C07332=1156.504,165.430,-58.579,-178.413,6.903,148.815
C07333=1156.500,165.680,-58.601,-178.411,6.904,148.815
C07334=1156.495,165.928,-58.623,-178.408,6.906,148.815
C07335=1156.491,166.178,-58.645,-178.405,6.909,148.814
C07336=1156.486,166.426,-58.667,-178.403,6.911,148.814
C07337=1156.481,166.675,-58.690,-178.400,6.913,148.814
C07338=1156.476,166.924,-58.711,-178.397,6.914,148.813
C07339=1156.472,167.173,-58.733,-178.394,6.917,148.813
C07340=1156.467,167.422,-58.755,-178.391,6.919,148.813
C07341=1156.463,167.671,-58.777,-178.389,6.920,148.812
C07342=1156.457,167.920,-58.799,-178.386,6.922,148.812
C07343=1156.453,168.169,-58.821,-178.383,6.925,148.812
C07344=1156.448,168.417,-58.844,-178.380,6.927,148.811
C07345=1156.444,168.667,-58.866,-178.378,6.928,148.811
C07346=1156.438,168.916,-58.888,-178.375,6.930,148.811
C07347=1156.434,169.165,-58.910,-178.372,6.933,148.811
C07348=1156.430,169.414,-58.932,-178.369,6.935,148.810
C07349=1156.425,169.662,-58.955,-178.367,6.937,148.810
C07350=1156.420,169.912,-58.977,-178.364,6.938,148.809
C07351=1156.415,170.161,-58.999,-178.361,6.941,148.809
C07352=1156.411,170.410,-59.021,-178.359,6.943,148.809
C07353=1156.407,170.658,-59.043,-178.356,6.945,148.809
C07354=1156.402,170.908,-59.066,-178.353,6.946,148.808
C07355=1156.397,171.157,-59.088,-178.350,6.949,148.808
C07356=1156.393,171.405,-59.111,-178.347,6.951,148.808
C07357=1156.388,171.655,-59.133,-178.345,6.953,148.807
C07358=1156.383,171.903,-59.155,-178.342,6.955,148.807
C07359=1156.379,172.152,-59.178,-178.339,6.957,148.807
C07360=1156.374,172.402,-59.200,-178.336,6.959,148.806
C07361=1156.369,172.650,-59.222,-178.334,6.961,148.806
C07362=1156.364,172.899,-59.245,-178.331,6.964,148.806
C07363=1156.359,173.148,-59.267,-178.328,6.965,148.805
C07364=1156.355,173.397,-59.290,-178.325,6.967,148.805
C07365=1156.350,173.646,-59.312,-178.322,6.970,148.805
C07366=1156.346,173.895,-59.334,-178.320,6.972,148.805
C07367=1156.341,174.144,-59.357,-178.317,6.973,148.804
C07368=1156.337,174.393,-59.379,-178.315,6.975,148.804
C07369=1156.332,174.642,-59.402,-178.311,6.978,148.803
C07370=1156.327,174.891,-59.425,-178.309,6.980,148.803
C07371=1156.323,175.140,-59.447,-178.306,6.982,148.803
C07372=1156.318,175.389,-59.470,-178.303,6.984,148.803
C07373=1156.314,175.638,-59.492,-178.300,6.986,148.802
C07374=1156.309,175.887,-59.515,-178.298,6.988,148.802
C07375=1156.304,176.135,-59.537,-178.295,6.991,148.802
C07376=1156.299,176.385,-59.560,-178.292,6.992,148.801
C07377=1156.295,176.634,-59.583,-178.290,6.994,148.801
C07378=1156.290,176.882,-59.606,-178.287,6.996,148.801
C07379=1156.285,177.131,-59.628,-178.284,6.999,148.801
C07380=1156.281,177.380,-59.651,-178.281,7.000,148.800
C07381=1156.276,177.630,-59.673,-178.279,7.002,148.800
C07382=1156.271,177.878,-59.696,-178.276,7.005,148.800
C07383=1156.267,178.127,-59.719,-178.273,7.007,148.799
C07384=1156.262,178.376,-59.742,-178.270,7.009,148.799
C07385=1156.258,178.624,-59.764,-178.268,7.012,148.799
C07386=1156.253,178.873,-59.787,-178.265,7.013,148.798
C07387=1156.249,179.123,-59.809,-178.262,7.015,148.798
C07388=1156.244,179.372,-59.833,-178.259,7.018,148.798
C07389=1156.239,179.620,-59.855,-178.257,7.020,148.798
C07390=1156.234,179.869,-59.878,-178.254,7.021,148.797
C07391=1156.230,180.118,-59.901,-178.251,7.024,148.797
C07392=1156.226,180.367,-59.924,-178.249,7.026,148.797
C07393=1156.221,180.616,-59.947,-178.246,7.028,148.796
C07394=1156.216,180.865,-59.969,-178.243,7.030,148.796
C07395=1156.211,181.114,-59.992,-178.240,7.032,148.796
C07396=1156.207,181.363,-60.016,-178.237,7.035,148.796
C07397=1156.203,181.612,-60.038,-178.235,7.037,148.795
C07398=1156.198,181.861,-60.062,-178.232,7.039,148.795
C07399=1156.193,182.110,-60.084,-178.229,7.041,148.795
C07400=1156.189,182.358,-60.107,-178.226,7.043,148.794
C07401=1156.184,182.607,-60.130,-178.224,7.045,148.794
C07402=1156.179,182.856,-60.154,-178.221,7.048,148.794
C07403=1156.175,183.105,-60.176,-178.218,7.050,148.794
C07404=1156.170,183.354,-60.200,-178.215,7.051,148.793
C07405=1156.165,183.624,-60.225,-178.212,7.054,148.793
C07406=1156.161,183.893,-60.249,-178.209,7.057,148.793
C07407=1156.155,184.163,-60.274,-178.207,7.059,148.792
C07408=1156.150,184.433,-60.299,-178.203,7.061,148.792
C07409=1156.145,184.682,-60.323,-178.201,7.063,148.792
C07410=1156.141,184.931,-60.345,-178.198,7.066,148.792
C07411=1156.136,185.179,-60.368,-178.195,7.068,148.791
C07412=1156.131,185.428,-60.392,-178.193,7.069,148.791
C07413=1156.127,185.677,-60.415,-178.190,7.072,148.791
C07414=1156.122,185.926,-60.438,-178.187,7.074,148.790
C07415=1156.118,186.175,-60.461,-178.184,7.077,148.790
C07416=1156.113,186.424,-60.485,-178.182,7.079,148.790
C07417=1156.109,186.673,-60.508,-178.179,7.080,148.790
C07418=1156.104,186.921,-60.532,-178.176,7.083,148.789
C07419=1156.099,187.170,-60.555,-178.173,7.085,148.789
C07420=1156.095,187.419,-60.578,-178.170,7.088,148.789
C07421=1156.090,187.667,-60.601,-178.168,7.089,148.788
C07422=1156.085,187.916,-60.625,-178.165,7.092,148.788
C07423=1156.081,188.165,-60.648,-178.162,7.094,148.788
C07424=1156.076,188.414,-60.671,-178.159,7.096,148.788
C07425=1156.071,188.664,-60.695,-178.157,7.099,148.787
C07426=1156.067,188.913,-60.718,-178.154,7.101,148.787
C07427=1156.062,189.161,-60.742,-178.151,7.102,148.787
C07428=1156.058,189.410,-60.765,-178.148,7.105,148.787
C07429=1156.054,189.659,-60.788,-178.146,7.107,148.786
C07430=1156.049,189.908,-60.811,-178.143,7.110,148.786
C07431=1156.044,190.157,-60.835,-178.140,7.112,148.786
C07432=1156.040,190.405,-60.859,-178.137,7.114,148.785
C07433=1156.035,190.654,-60.882,-178.135,7.116,148.785
C07434=1156.030,190.903,-60.906,-178.132,7.118,148.785
C07435=1156.026,191.152,-60.929,-178.129,7.121,148.785
C07436=1156.021,191.401,-60.953,-178.127,7.123,148.784
C07437=1156.017,191.650,-60.976,-178.123,7.125,148.784
C07438=1156.012,191.899,-61.000,-178.121,7.127,148.784
C07439=1156.008,192.147,-61.024,-178.118,7.129,148.784
C07440=1156.003,192.396,-61.047,-178.115,7.132,148.783
C07441=1155.998,192.645,-61.071,-178.113,7.134,148.783
C07442=1155.994,192.894,-61.095,-178.110,7.136,148.783
C07443=1155.989,193.143,-61.118,-178.107,7.138,148.783
C07444=1155.984,193.392,-61.141,-178.104,7.141,148.782
C07445=1155.980,193.640,-61.165,-178.102,7.143,148.782
C07446=1155.975,193.889,-61.189,-178.099,7.146,148.782
C07447=1155.971,194.138,-61.212,-178.096,7.147,148.782
C07448=1155.966,194.387,-61.236,-178.094,7.150,148.781
C07449=1155.961,194.636,-61.260,-178.091,7.152,148.781
C07450=1155.957,194.884,-61.284,-178.088,7.154,148.781
C07451=1155.952,195.133,-61.307,-178.085,7.157,148.781
C07452=1155.947,195.382,-61.332,-178.082,7.159,148.780
C07453=1155.943,195.632,-61.355,-178.080,7.162,148.780
C07454=1155.939,195.880,-61.380,-178.077,7.163,148.780
C07455=1155.934,196.129,-61.403,-178.074,7.166,148.780
C07456=1155.930,196.377,-61.427,-178.071,7.168,148.779
C07457=1155.925,196.626,-61.450,-178.068,7.171,148.779
C07458=1155.921,196.875,-61.474,-178.066,7.173,148.779
C07459=1155.916,197.124,-61.498,-178.063,7.175,148.779
C07460=1155.911,197.373,-61.522,-178.061,7.177,148.778
C07461=1155.906,197.621,-61.546,-178.058,7.179,148.778
C07462=1155.902,197.871,-61.570,-178.055,7.182,148.778
C07463=1155.898,198.119,-61.594,-178.052,7.184,148.778
C07464=1155.893,198.368,-61.618,-178.049,7.186,148.777
C07465=1155.889,198.617,-61.642,-178.047,7.188,148.777
C07466=1155.884,198.865,-61.666,-178.044,7.191,148.777
C07467=1155.879,199.114,-61.690,-178.041,7.193,148.777
C07468=1155.875,199.363,-61.714,-178.038,7.196,148.776
C07469=1155.871,199.612,-61.738,-178.036,7.198,148.776
C07470=1155.865,199.861,-61.762,-178.033,7.200,148.776
C07471=1155.861,200.110,-61.786,-178.030,7.202,148.776
C07472=1155.856,200.358,-61.810,-178.027,7.205,148.776
C07473=1155.852,200.606,-61.834,-178.025,7.207,148.775
C07474=1155.847,200.857,-61.859,-178.022,7.210,148.775
C07475=1155.843,201.105,-61.883,-178.019,7.211,148.775
C07476=1155.838,201.353,-61.907,-178.016,7.214,148.775
C07477=1155.834,201.602,-61.931,-178.014,7.216,148.774
C07478=1155.829,201.851,-61.955,-178.011,7.219,148.774
C07479=1155.825,202.100,-61.979,-178.008,7.221,148.774
C07480=1155.820,202.349,-62.003,-178.005,7.224,148.774
C07481=1155.815,202.597,-62.028,-178.003,7.226,148.773
C07482=1155.811,202.846,-62.052,-178.000,7.228,148.773
C07483=1155.807,203.095,-62.077,-177.997,7.230,148.773
C07484=1155.802,203.344,-62.101,-177.994,7.233,148.773
C07485=1155.797,203.593,-62.125,-177.992,7.235,148.772
C07486=1155.793,203.841,-62.149,-177.989,7.238,148.772
C07487=1155.788,204.090,-62.174,-177.986,7.240,148.772
C07488=1155.784,204.339,-62.198,-177.983,7.242,148.772
C07489=1155.779,204.588,-62.223,-177.981,7.244,148.772
C07490=1155.774,204.836,-62.247,-177.978,7.247,148.771
C07491=1155.771,205.085,-62.271,-177.975,7.250,148.771
C07492=1155.766,205.334,-62.296,-177.973,7.252,148.771
C07493=1155.761,205.582,-62.320,-177.969,7.254,148.771
C07494=1155.757,205.832,-62.345,-177.967,7.257,148.771
C07495=1155.752,206.080,-62.369,-177.964,7.259,148.770
C07496=1155.747,206.329,-62.394,-177.962,7.261,148.770
C07497=1155.743,206.577,-62.418,-177.958,7.264,148.770
C07498=1155.738,206.827,-62.443,-177.956,7.266,148.770
C07499=1155.734,207.075,-62.467,-177.953,7.269,148.769
C07500=1155.729,207.324,-62.491,-177.951,7.271,148.769
C07501=1155.725,207.573,-62.516,-177.947,7.273,148.769
C07502=1155.720,207.822,-62.541,-177.945,7.275,148.769
C07503=1155.715,208.070,-62.565,-177.942,7.278,148.769
C07504=1155.711,208.319,-62.590,-177.939,7.281,148.768
C07505=1155.706,208.568,-62.614,-177.937,7.283,148.768
C07506=1155.702,208.816,-62.639,-177.934,7.285,148.768
C07507=1155.698,209.065,-62.664,-177.931,7.288,148.768
C07508=1155.693,209.314,-62.688,-177.928,7.290,148.767
C07509=1155.688,209.585,-62.715,-177.925,7.293,148.767
C07510=1155.683,209.855,-62.742,-177.922,7.296,148.767
C07511=1155.678,210.126,-62.769,-177.920,7.298,148.767
C07512=1155.673,210.396,-62.796,-177.917,7.300,148.767
C07513=1155.668,210.645,-62.820,-177.914,7.303,148.767
C07514=1155.664,210.894,-62.845,-177.911,7.305,148.766
C07515=1155.659,211.142,-62.870,-177.908,7.308,148.766
C07516=1155.655,211.391,-62.895,-177.905,7.311,148.766
C07517=1155.651,211.640,-62.919,-177.903,7.313,148.766
C07518=1155.645,211.888,-62.944,-177.900,7.315,148.765
C07519=1155.642,212.137,-62.969,-177.898,7.317,148.765
C07520=1155.637,212.386,-62.994,-177.894,7.320,148.765
C07521=1155.632,212.635,-63.019,-177.891,7.323,148.765
C07522=1155.628,212.883,-63.044,-177.889,7.325,148.765
C07523=1155.624,213.132,-63.069,-177.886,7.328,148.764
C07524=1155.619,213.381,-63.093,-177.884,7.330,148.764
C07525=1155.614,213.630,-63.119,-177.881,7.332,148.764
C07526=1155.610,213.878,-63.143,-177.878,7.334,148.764
C07527=1155.605,214.127,-63.168,-177.876,7.337,148.764
C07528=1155.601,214.376,-63.194,-177.872,7.340,148.763
C07529=1155.596,214.624,-63.218,-177.870,7.342,148.763
C07530=1155.592,214.873,-63.243,-177.867,7.345,148.763
C07531=1155.587,215.122,-63.268,-177.865,7.347,148.763
C07532=1155.583,215.371,-63.294,-177.862,7.350,148.763
C07533=1155.578,215.619,-63.318,-177.859,7.352,148.762
C07534=1155.574,215.868,-63.344,-177.856,7.354,148.762
C07535=1155.569,216.116,-63.368,-177.853,7.357,148.762
C07536=1155.565,216.365,-63.394,-177.850,7.360,148.762
C07537=1155.560,216.614,-63.418,-177.848,7.362,148.762
C07538=1155.556,216.862,-63.444,-177.845,7.365,148.761
C07539=1155.551,217.112,-63.469,-177.843,7.367,148.761
C07540=1155.547,217.360,-63.494,-177.839,7.369,148.761
C07541=1155.542,217.609,-63.520,-177.837,7.372,148.761
C07542=1155.537,217.858,-63.545,-177.834,7.374,148.761
C07543=1155.534,218.106,-63.570,-177.831,7.377,148.761
C07544=1155.529,218.355,-63.595,-177.828,7.380,148.760
C07545=1155.524,218.604,-63.620,-177.826,7.382,148.760
C07546=1155.520,218.852,-63.646,-177.823,7.384,148.760
C07547=1155.515,219.101,-63.671,-177.821,7.387,148.760
C07548=1155.511,219.350,-63.697,-177.818,7.390,148.760
C07549=1155.506,219.598,-63.722,-177.815,7.392,148.759
C07550=1155.501,219.847,-63.747,-177.813,7.394,148.759
C07551=1155.497,220.095,-63.772,-177.809,7.397,148.759
C07552=1155.493,220.344,-63.798,-177.806,7.400,148.759
C07553=1155.489,220.593,-63.823,-177.804,7.402,148.759
C07554=1155.484,220.842,-63.848,-177.801,7.404,148.759
C07555=1155.480,221.090,-63.874,-177.798,7.407,148.758
C07556=1155.475,221.338,-63.899,-177.796,7.409,148.758
C07557=1155.471,221.587,-63.925,-177.793,7.412,148.758
C07558=1155.466,221.837,-63.950,-177.790,7.415,148.758
C07559=1155.461,222.085,-63.975,-177.788,7.417,148.758
C07560=1155.457,222.334,-64.001,-177.785,7.420,148.758
C07561=1155.453,222.582,-64.027,-177.782,7.423,148.757
C07562=1155.448,222.830,-64.052,-177.780,7.425,148.757
C07563=1155.444,223.079,-64.078,-177.776,7.427,148.757
C07564=1155.439,223.329,-64.103,-177.774,7.430,148.757
C07565=1155.434,223.577,-64.128,-177.771,7.432,148.757
C07566=1155.430,223.826,-64.154,-177.768,7.435,148.756
C07567=1155.426,224.074,-64.180,-177.765,7.438,148.756
C07568=1155.421,224.323,-64.205,-177.763,7.440,148.756
C07569=1155.417,224.571,-64.231,-177.760,7.443,148.756
C07570=1155.413,224.820,-64.257,-177.757,7.446,148.756
C07571=1155.407,225.069,-64.283,-177.755,7.448,148.756
C07572=1155.403,225.317,-64.308,-177.752,7.451,148.756
C07573=1155.399,225.566,-64.334,-177.749,7.453,148.755
C07574=1155.394,225.814,-64.360,-177.747,7.455,148.755
C07575=1155.390,226.063,-64.385,-177.744,7.458,148.755
C07576=1155.385,226.312,-64.411,-177.741,7.461,148.755
C07577=1155.381,226.561,-64.437,-177.738,7.464,148.755
C07578=1155.376,226.809,-64.462,-177.736,7.466,148.755
C07579=1155.372,227.058,-64.488,-177.732,7.468,148.754
C07580=1155.367,227.307,-64.514,-177.730,7.471,148.754
C07581=1155.363,227.556,-64.540,-177.727,7.473,148.754
C07582=1155.358,227.804,-64.565,-177.725,7.476,148.754
C07583=1155.354,228.052,-64.592,-177.721,7.479,148.754
C07584=1155.350,228.301,-64.618,-177.719,7.481,148.754
C07585=1155.345,228.550,-64.644,-177.716,7.484,148.754
C07586=1155.340,228.798,-64.669,-177.713,7.487,148.753
C07587=1155.336,229.047,-64.695,-177.710,7.490,148.753
C07588=1155.332,229.295,-64.721,-177.708,7.492,148.753
C07589=1155.328,229.544,-64.747,-177.705,7.495,148.753
C07590=1155.323,229.793,-64.774,-177.702,7.497,148.753
C07591=1155.318,230.041,-64.799,-177.699,7.500,148.753
C07592=1155.314,230.290,-64.825,-177.697,7.502,148.753
C07593=1155.309,230.538,-64.851,-177.694,7.505,148.752
C07594=1155.305,230.787,-64.878,-177.691,7.508,148.752
C07595=1155.301,231.036,-64.903,-177.689,7.510,148.752
C07596=1155.296,231.285,-64.929,-177.686,7.513,148.752
C07597=1155.291,231.532,-64.956,-177.683,7.516,148.752
C07598=1155.287,231.781,-64.982,-177.680,7.518,148.752
C07599=1155.283,232.030,-65.007,-177.678,7.520,148.751
C07600=1155.278,232.278,-65.034,-177.675,7.523,148.751
C07601=1155.274,232.527,-65.060,-177.672,7.526,148.751
C07602=1155.270,232.776,-65.086,-177.669,7.529,148.751
C07603=1155.264,233.024,-65.113,-177.667,7.531,148.751
C07604=1155.260,233.273,-65.138,-177.664,7.534,148.751
C07605=1155.256,233.521,-65.164,-177.661,7.537,148.751
C07606=1155.251,233.770,-65.191,-177.659,7.540,148.751
C07607=1155.247,234.019,-65.217,-177.656,7.542,148.750
C07608=1155.242,234.267,-65.244,-177.653,7.545,148.750
C07609=1155.238,234.516,-65.270,-177.650,7.547,148.750
C07610=1155.234,234.764,-65.296,-177.648,7.550,148.750
C07611=1155.229,235.013,-65.323,-177.645,7.552,148.750
C07612=1155.225,235.262,-65.349,-177.642,7.555,148.750
C07613=1155.220,235.534,-65.378,-177.639,7.558,148.750
C07614=1155.215,235.805,-65.406,-177.637,7.561,148.749
C07615=1155.210,236.077,-65.435,-177.633,7.564,148.749
C07616=1155.206,236.349,-65.464,-177.630,7.567,148.749
C07617=1155.201,236.597,-65.491,-177.628,7.569,148.749
C07618=1155.197,236.846,-65.517,-177.625,7.572,148.749
C07619=1155.192,237.094,-65.544,-177.622,7.575,148.749
C07620=1155.188,237.343,-65.569,-177.619,7.578,148.749
C07621=1155.183,237.592,-65.596,-177.616,7.581,148.749
C07622=1155.179,237.840,-65.623,-177.614,7.583,148.748
C07623=1155.174,238.089,-65.649,-177.611,7.586,148.748
C07624=1155.170,238.337,-65.676,-177.608,7.589,148.748
C07625=1155.166,238.586,-65.703,-177.605,7.591,148.748
C07626=1155.161,238.835,-65.729,-177.603,7.594,148.748
C07627=1155.157,239.083,-65.756,-177.600,7.596,148.748
C07628=1155.152,239.331,-65.783,-177.597,7.599,148.748
C07629=1155.148,239.580,-65.808,-177.595,7.602,148.748
C07630=1155.143,239.829,-65.835,-177.591,7.605,148.747
C07631=1155.139,240.077,-65.862,-177.589,7.607,148.747
C07632=1155.135,240.325,-65.889,-177.586,7.610,148.747
C07633=1155.130,240.574,-65.916,-177.584,7.613,148.747
C07634=1155.126,240.823,-65.942,-177.581,7.616,148.747
C07635=1155.121,241.071,-65.969,-177.578,7.619,148.747
C07636=1155.117,241.320,-65.996,-177.575,7.621,148.747
C07637=1155.113,241.568,-66.022,-177.573,7.624,148.747
C07638=1155.108,241.816,-66.049,-177.570,7.626,148.746
C07639=1155.103,242.065,-66.076,-177.567,7.629,148.746
C07640=1155.099,242.314,-66.102,-177.564,7.632,148.746
C07641=1155.094,242.562,-66.129,-177.562,7.635,148.746
C07642=1155.090,242.811,-66.156,-177.559,7.637,148.746
C07643=1155.086,243.059,-66.183,-177.556,7.640,148.746
C07644=1155.081,243.307,-66.210,-177.553,7.643,148.746
C07645=1155.077,243.556,-66.237,-177.551,7.646,148.746
C07646=1155.073,243.804,-66.263,-177.548,7.649,148.746
C07647=1155.069,244.053,-66.291,-177.546,7.651,148.746
C07648=1155.064,244.302,-66.318,-177.543,7.654,148.745
C07649=1155.059,244.550,-66.345,-177.540,7.657,148.745
C07650=1155.055,244.798,-66.371,-177.537,7.660,148.745
C07651=1155.051,245.047,-66.399,-177.534,7.663,148.745
C07652=1155.046,245.295,-66.426,-177.531,7.665,148.745
C07653=1155.041,245.544,-66.453,-177.529,7.667,148.745
C07654=1155.037,245.792,-66.479,-177.526,7.670,148.745
C07655=1155.033,246.041,-66.507,-177.523,7.673,148.745
C07656=1155.029,246.290,-66.534,-177.521,7.676,148.745
C07657=1155.024,246.538,-66.561,-177.518,7.679,148.745
C07658=1155.019,246.787,-66.588,-177.515,7.682,148.744
C07659=1155.015,247.035,-66.615,-177.512,7.685,148.744
C07660=1155.011,247.283,-66.641,-177.510,7.687,148.744
C07661=1155.007,247.532,-66.669,-177.507,7.690,148.744
C07662=1155.002,247.781,-66.696,-177.504,7.693,148.744
C07663=1154.998,248.029,-66.724,-177.501,7.696,148.744
C07664=1154.993,248.277,-66.751,-177.499,7.699,148.744
C07665=1154.989,248.526,-66.778,-177.496,7.702,148.744
C07666=1154.984,248.774,-66.805,-177.494,7.704,148.744
C07667=1154.980,249.023,-66.833,-177.491,7.707,148.744
C07668=1154.975,249.272,-66.860,-177.488,7.709,148.744
C07669=1154.972,249.520,-66.886,-177.485,7.712,148.743
C07670=1154.967,249.768,-66.913,-177.483,7.715,148.743
C07671=1154.963,250.017,-66.942,-177.480,7.718,148.743
C07672=1154.958,250.265,-66.969,-177.477,7.721,148.743
C07673=1154.954,250.514,-66.996,-177.474,7.724,148.743
C07674=1154.949,250.762,-67.023,-177.472,7.726,148.743
C07675=1154.945,251.011,-67.051,-177.469,7.729,148.743
C07676=1154.941,251.259,-67.078,-177.466,7.732,148.743
C07677=1154.936,251.507,-67.106,-177.464,7.735,148.743
C07678=1154.932,251.756,-67.133,-177.460,7.738,148.743
C07679=1154.928,252.005,-67.160,-177.458,7.741,148.743
C07680=1154.923,252.253,-67.188,-177.455,7.744,148.742
C07681=1154.919,252.501,-67.215,-177.452,7.747,148.742
C07682=1154.914,252.749,-67.243,-177.450,7.749,148.742
C07683=1154.910,252.998,-67.270,-177.447,7.752,148.742
C07684=1154.906,253.247,-67.297,-177.444,7.755,148.742
C07685=1154.901,253.495,-67.325,-177.442,7.757,148.742
C07686=1154.897,253.744,-67.353,-177.439,7.760,148.742
C07687=1154.893,253.992,-67.380,-177.436,7.763,148.742
C07688=1154.887,254.241,-67.408,-177.433,7.766,148.742
C07689=1154.884,254.489,-67.436,-177.431,7.769,148.742
C07690=1154.879,254.738,-67.463,-177.428,7.772,148.742
C07691=1154.875,254.986,-67.491,-177.426,7.774,148.742
C07692=1154.871,255.234,-67.519,-177.423,7.777,148.742
C07693=1154.866,255.483,-67.546,-177.420,7.780,148.742
C07694=1154.862,255.731,-67.574,-177.417,7.783,148.741
C07695=1154.858,255.980,-67.601,-177.414,7.786,148.741
C07696=1154.853,256.228,-67.630,-177.412,7.789,148.741
C07697=1154.848,256.476,-67.657,-177.409,7.792,148.741
C07698=1154.844,256.725,-67.685,-177.406,7.795,148.741
C07699=1154.840,256.973,-67.713,-177.403,7.798,148.741
C07700=1154.836,257.222,-67.740,-177.401,7.801,148.741
C07701=1154.832,257.470,-67.768,-177.398,7.804,148.741
C07702=1154.827,257.718,-67.796,-177.396,7.806,148.741
C07703=1154.822,257.967,-67.824,-177.393,7.809,148.741
C07704=1154.818,258.215,-67.852,-177.390,7.812,148.741
C07705=1154.814,258.464,-67.880,-177.387,7.815,148.741
C07706=1154.809,258.712,-67.908,-177.385,7.818,148.741
C07707=1154.805,258.960,-67.935,-177.382,7.821,148.741
C07708=1154.801,259.209,-67.963,-177.379,7.823,148.741
C07709=1154.797,259.457,-67.991,-177.377,7.827,148.741
C07710=1154.792,259.706,-68.020,-177.374,7.830,148.741
C07711=1154.788,259.954,-68.048,-177.371,7.833,148.741
C07712=1154.784,260.203,-68.075,-177.368,7.836,148.741
C07713=1154.779,260.451,-68.103,-177.366,7.839,148.740
C07714=1154.774,260.699,-68.131,-177.363,7.841,148.740
C07715=1154.770,260.947,-68.159,-177.360,7.844,148.740
C07716=1154.766,261.195,-68.187,-177.358,7.847,148.740
C07717=1154.761,261.469,-68.218,-177.355,7.850,148.740
C07718=1154.756,261.742,-68.249,-177.352,7.853,148.740
C07719=1154.751,262.016,-68.280,-177.349,7.856,148.740
C07720=1154.747,262.289,-68.310,-177.346,7.860,148.740
C07721=1154.742,262.538,-68.339,-177.343,7.863,148.740
C07722=1154.738,262.786,-68.367,-177.340,7.866,148.740
C07723=1154.733,263.035,-68.396,-177.337,7.869,148.740
C07724=1154.729,263.283,-68.423,-177.335,7.872,148.740
C07725=1154.725,263.531,-68.452,-177.332,7.875,148.740
C07726=1154.720,263.779,-68.480,-177.329,7.878,148.740
C07727=1154.716,264.028,-68.508,-177.327,7.880,148.740
C07728=1154.712,264.277,-68.537,-177.324,7.883,148.740
C07729=1154.708,264.525,-68.565,-177.322,7.886,148.740
C07730=1154.703,264.774,-68.593,-177.319,7.889,148.740
C07731=1154.699,265.021,-68.622,-177.316,7.892,148.740
C07732=1154.695,265.270,-68.651,-177.313,7.895,148.740
C07733=1154.690,265.518,-68.678,-177.311,7.898,148.740
C07734=1154.686,265.766,-68.707,-177.308,7.901,148.739
C07735=1154.681,266.014,-68.735,-177.305,7.904,148.739
C07736=1154.677,266.263,-68.764,-177.302,7.907,148.739
C07737=1154.673,266.512,-68.792,-177.300,7.910,148.740
C07738=1154.668,266.760,-68.820,-177.297,7.913,148.739
C07739=1154.665,267.008,-68.849,-177.294,7.916,148.739
C07740=1154.660,267.256,-68.877,-177.292,7.919,148.739
C07741=1154.656,267.505,-68.905,-177.289,7.922,148.739
C07742=1154.651,267.753,-68.934,-177.286,7.925,148.739
C07743=1154.647,268.001,-68.963,-177.283,7.927,148.739
C07744=1154.643,268.250,-68.991,-177.281,7.930,148.739
C07745=1154.638,268.498,-69.020,-177.278,7.934,148.739
C07746=1154.634,268.746,-69.048,-177.276,7.937,148.739
C07747=1154.630,268.995,-69.077,-177.273,7.940,148.739
C07748=1154.625,269.243,-69.105,-177.270,7.943,148.739
C07749=1154.621,269.492,-69.134,-177.267,7.945,148.739
C07750=1154.617,269.740,-69.163,-177.264,7.948,148.739
C07751=1154.612,269.988,-69.191,-177.262,7.952,148.739
C07752=1154.608,270.237,-69.220,-177.259,7.955,148.739
C07753=1154.604,270.485,-69.249,-177.257,7.958,148.739
C07754=1154.599,270.733,-69.277,-177.254,7.961,148.739
C07755=1154.595,270.981,-69.307,-177.251,7.963,148.739
C07756=1154.591,271.230,-69.335,-177.248,7.966,148.739
C07757=1154.586,271.478,-69.363,-177.246,7.970,148.739
C07758=1154.582,271.726,-69.392,-177.243,7.973,148.739
C07759=1154.578,271.975,-69.421,-177.240,7.976,148.739
C07760=1154.574,272.222,-69.450,-177.238,7.979,148.739
C07761=1154.569,272.471,-69.478,-177.235,7.981,148.739
C07762=1154.565,272.719,-69.508,-177.233,7.985,148.739
C07763=1154.560,272.968,-69.537,-177.230,7.988,148.739
C07764=1154.556,273.215,-69.565,-177.227,7.991,148.739
C07765=1154.552,273.464,-69.594,-177.224,7.994,148.739
C07766=1154.548,273.713,-69.623,-177.221,7.997,148.739
C07767=1154.543,273.961,-69.652,-177.219,8.000,148.739
C07768=1154.539,274.209,-69.681,-177.216,8.003,148.739
C07769=1154.535,274.457,-69.710,-177.214,8.006,148.739
C07770=1154.531,274.706,-69.739,-177.211,8.009,148.739
C07771=1154.526,274.954,-69.768,-177.208,8.012,148.739
C07772=1154.521,275.202,-69.797,-177.206,8.015,148.739
C07773=1154.518,275.450,-69.825,-177.203,8.018,148.739
C07774=1154.514,275.699,-69.855,-177.200,8.021,148.739
C07775=1154.509,275.947,-69.884,-177.197,8.024,148.739
C07776=1154.504,276.195,-69.913,-177.195,8.027,148.739
C07777=1154.500,276.443,-69.942,-177.192,8.030,148.739
C07778=1154.496,276.692,-69.972,-177.190,8.033,148.739
C07779=1154.492,276.940,-70.000,-177.187,8.036,148.739
C07780=1154.488,277.188,-70.029,-177.185,8.039,148.739
C07781=1154.483,277.436,-70.058,-177.182,8.042,148.739
C07782=1154.479,277.684,-70.088,-177.179,8.045,148.739
C07783=1154.475,277.933,-70.116,-177.176,8.048,148.739
C07784=1154.470,278.181,-70.146,-177.174,8.051,148.739
C07785=1154.466,278.430,-70.175,-177.171,8.055,148.739
C07786=1154.462,278.678,-70.205,-177.168,8.058,148.739
C07787=1154.458,278.926,-70.234,-177.165,8.061,148.739
C07788=1154.453,279.174,-70.263,-177.163,8.064,148.739
C07789=1154.449,279.423,-70.292,-177.160,8.067,148.739
C07790=1154.444,279.671,-70.322,-177.157,8.070,148.739
C07791=1154.440,279.919,-70.351,-177.154,8.073,148.739
C07792=1154.436,280.167,-70.380,-177.152,8.076,148.739
C07793=1154.432,280.416,-70.410,-177.149,8.079,148.739
C07794=1154.428,280.664,-70.439,-177.147,8.082,148.739
C07795=1154.424,280.912,-70.469,-177.144,8.085,148.739
C07796=1154.419,281.160,-70.498,-177.142,8.088,148.739
C07797=1154.415,281.408,-70.527,-177.139,8.091,148.739
C07798=1154.410,281.656,-70.557,-177.136,8.095,148.739
C07799=1154.406,281.905,-70.586,-177.134,8.098,148.739
C07800=1154.402,282.153,-70.616,-177.131,8.101,148.739
C07801=1154.398,282.401,-70.645,-177.128,8.103,148.739
C07802=1154.394,282.649,-70.675,-177.126,8.107,148.739
C07803=1154.390,282.898,-70.704,-177.122,8.111,148.739
C07804=1154.385,283.146,-70.734,-177.120,8.113,148.739
C07805=1154.380,283.395,-70.764,-177.117,8.117,148.739
C07806=1154.376,283.643,-70.793,-177.115,8.120,148.739
C07807=1154.372,283.891,-70.823,-177.112,8.123,148.739
C07808=1154.368,284.139,-70.852,-177.110,8.126,148.739
C07809=1154.364,284.387,-70.882,-177.107,8.129,148.739
C07810=1154.360,284.635,-70.912,-177.104,8.132,148.739
C07811=1154.356,284.884,-70.941,-177.102,8.135,148.740
C07812=1154.350,285.131,-70.971,-177.099,8.138,148.740
C07813=1154.346,285.380,-71.000,-177.096,8.141,148.739
C07814=1154.342,285.628,-71.030,-177.094,8.144,148.740
C07815=1154.338,285.876,-71.060,-177.091,8.148,148.740
C07816=1154.334,286.124,-71.089,-177.088,8.151,148.740
C07817=1154.329,286.372,-71.119,-177.085,8.154,148.740
C07818=1154.325,286.621,-71.149,-177.083,8.157,148.740
C07819=1154.321,286.869,-71.179,-177.080,8.160,148.740
C07820=1154.317,287.117,-71.209,-177.078,8.163,148.740
C07821=1154.312,287.392,-71.242,-177.074,8.167,148.740
C07822=1154.308,287.667,-71.275,-177.072,8.170,148.740
C07823=1154.303,287.942,-71.308,-177.069,8.174,148.740
C07824=1154.297,288.218,-71.341,-177.066,8.177,148.740
C07825=1154.293,288.466,-71.371,-177.064,8.180,148.740
C07826=1154.289,288.714,-71.401,-177.061,8.183,148.740
C07827=1154.285,288.962,-71.430,-177.058,8.186,148.740
C07828=1154.281,289.211,-71.461,-177.055,8.190,148.740
C07829=1154.277,289.459,-71.491,-177.052,8.193,148.740
C07830=1154.273,289.707,-71.521,-177.050,8.197,148.740
C07831=1154.268,289.955,-71.551,-177.047,8.200,148.740
C07832=1154.264,290.203,-71.581,-177.044,8.203,148.740
C07833=1154.260,290.451,-71.611,-177.042,8.206,148.741
C07834=1154.255,290.700,-71.641,-177.039,8.209,148.740
C07835=1154.251,290.947,-71.671,-177.037,8.212,148.741
C07836=1154.247,291.195,-71.702,-177.034,8.215,148.741
C07837=1154.242,291.444,-71.731,-177.031,8.219,148.741
C07838=1154.239,291.692,-71.762,-177.029,8.222,148.741
C07839=1154.234,291.941,-71.792,-177.026,8.225,148.741
C07840=1154.230,292.188,-71.822,-177.024,8.228,148.741
C07841=1154.225,292.437,-71.852,-177.021,8.231,148.741
C07842=1154.221,292.684,-71.882,-177.019,8.235,148.741
C07843=1154.218,292.932,-71.912,-177.016,8.237,148.741
C07844=1154.213,293.181,-71.943,-177.013,8.241,148.741
C07845=1154.209,293.429,-71.973,-177.010,8.245,148.741
C07846=1154.205,293.678,-72.003,-177.008,8.248,148.741
C07847=1154.201,293.925,-72.033,-177.005,8.251,148.741
C07848=1154.196,294.173,-72.064,-177.002,8.254,148.741
C07849=1154.192,294.421,-72.094,-177.000,8.257,148.741
C07850=1154.188,294.670,-72.124,-176.997,8.260,148.741
C07851=1154.184,294.918,-72.155,-176.995,8.263,148.742
C07852=1154.179,295.166,-72.185,-176.992,8.267,148.742
C07853=1154.175,295.414,-72.215,-176.989,8.270,148.742
C07854=1154.171,295.662,-72.246,-176.986,8.273,148.742
C07855=1154.167,295.910,-72.276,-176.984,8.276,148.742
C07856=1154.163,296.158,-72.307,-176.981,8.279,148.742
C07857=1154.158,296.406,-72.338,-176.979,8.283,148.742
C07858=1154.154,296.654,-72.367,-176.976,8.286,148.742
C07859=1154.150,296.903,-72.398,-176.973,8.290,148.742
C07860=1154.146,297.151,-72.428,-176.971,8.293,148.742
C07861=1154.141,297.399,-72.459,-176.968,8.296,148.742
C07862=1154.137,297.647,-72.490,-176.966,8.299,148.742
C07863=1154.133,297.895,-72.520,-176.963,8.302,148.743
C07864=1154.129,298.143,-72.551,-176.960,8.305,148.743
C07865=1154.125,298.391,-72.581,-176.958,8.309,148.743
C07866=1154.120,298.639,-72.611,-176.955,8.312,148.743
C07867=1154.116,298.888,-72.643,-176.953,8.315,148.743
C07868=1154.112,299.136,-72.673,-176.950,8.318,148.743
C07869=1154.108,299.383,-72.703,-176.947,8.322,148.743
C07870=1154.104,299.632,-72.735,-176.945,8.325,148.743
C07871=1154.100,299.880,-72.765,-176.942,8.329,148.743
C07872=1154.095,300.128,-72.796,-176.939,8.332,148.743
C07873=1154.090,300.376,-72.826,-176.937,8.335,148.743
C07874=1154.086,300.624,-72.857,-176.934,8.338,148.744
C07875=1154.083,300.872,-72.888,-176.932,8.341,148.744
C07876=1154.078,301.119,-72.919,-176.929,8.344,148.744
C07877=1154.074,301.368,-72.950,-176.926,8.348,148.744
C07878=1154.070,301.616,-72.981,-176.924,8.352,148.744
C07879=1154.066,301.864,-73.011,-176.921,8.354,148.744
C07880=1154.062,302.112,-73.042,-176.919,8.358,148.744
C07881=1154.057,302.360,-73.073,-176.916,8.361,148.744
C07882=1154.053,302.609,-73.104,-176.913,8.365,148.744
C07883=1154.048,302.857,-73.135,-176.911,8.368,148.744
C07884=1154.045,303.104,-73.166,-176.908,8.371,148.744
C07885=1154.041,303.353,-73.197,-176.906,8.374,148.745
C07886=1154.036,303.600,-73.228,-176.903,8.378,148.745
C07887=1154.032,303.848,-73.258,-176.900,8.381,148.745
C07888=1154.028,304.097,-73.290,-176.898,8.385,148.745
C07889=1154.023,304.344,-73.321,-176.895,8.388,148.745
C07890=1154.019,304.593,-73.352,-176.892,8.391,148.745
C07891=1154.015,304.841,-73.382,-176.890,8.394,148.745
C07892=1154.011,305.089,-73.413,-176.887,8.398,148.745
C07893=1154.007,305.337,-73.445,-176.885,8.401,148.745
C07894=1154.003,305.585,-73.476,-176.882,8.404,148.745
C07895=1153.999,305.833,-73.507,-176.879,8.407,148.746
C07896=1153.994,306.081,-73.538,-176.877,8.411,148.746
C07897=1153.990,306.329,-73.569,-176.874,8.414,148.746
C07898=1153.986,306.577,-73.601,-176.871,8.418,148.746
C07899=1153.981,306.825,-73.632,-176.869,8.421,148.746
C07900=1153.977,307.073,-73.663,-176.866,8.424,148.746
C07901=1153.973,307.321,-73.694,-176.864,8.427,148.746
C07902=1153.969,307.569,-73.725,-176.861,8.431,148.746
C07903=1153.965,307.817,-73.757,-176.858,8.434,148.747
C07904=1153.961,308.065,-73.788,-176.856,8.438,148.747
C07905=1153.956,308.313,-73.820,-176.853,8.441,148.747
C07906=1153.952,308.561,-73.851,-176.851,8.444,148.747
C07907=1153.948,308.809,-73.882,-176.848,8.448,148.747
C07908=1153.944,309.057,-73.913,-176.845,8.451,148.747
C07909=1153.940,309.305,-73.945,-176.843,8.454,148.747
C07910=1153.936,309.553,-73.976,-176.841,8.457,148.747
C07911=1153.931,309.801,-74.007,-176.837,8.461,148.747
C07912=1153.927,310.049,-74.039,-176.835,8.464,148.748
C07913=1153.923,310.297,-74.070,-176.833,8.468,148.748
C07914=1153.919,310.545,-74.101,-176.830,8.471,148.748
C07915=1153.915,310.793,-74.133,-176.827,8.475,148.748
C07916=1153.911,311.041,-74.164,-176.825,8.478,148.748
C07917=1153.906,311.289,-74.195,-176.822,8.481,148.748
C07918=1153.903,311.537,-74.227,-176.820,8.484,148.748
C07919=1153.898,311.784,-74.259,-176.817,8.488,148.749
C07920=1153.894,312.033,-74.290,-176.814,8.491,148.749
C07921=1153.890,312.281,-74.322,-176.812,8.495,148.749
C07922=1153.886,312.528,-74.354,-176.809,8.498,148.749
C07923=1153.882,312.777,-74.385,-176.807,8.502,148.749
C07924=1153.877,313.024,-74.416,-176.804,8.505,148.749
C07925=1153.873,313.302,-74.452,-176.801,8.509,148.749
C07926=1153.869,313.579,-74.487,-176.799,8.512,148.750
C07927=1153.863,313.857,-74.523,-176.795,8.516,148.750
C07928=1153.858,314.135,-74.558,-176.792,8.520,148.750
C07929=1153.855,314.383,-74.590,-176.790,8.523,148.750
C07930=1153.850,314.630,-74.621,-176.788,8.527,148.750
C07931=1153.847,314.878,-74.653,-176.784,8.531,148.750
C07932=1153.842,315.126,-74.686,-176.782,8.534,148.750
C07933=1153.838,315.374,-74.717,-176.780,8.537,148.751
C07934=1153.834,315.622,-74.749,-176.777,8.540,148.751
C07935=1153.830,315.870,-74.780,-176.774,8.544,148.751
C07936=1153.825,316.118,-74.812,-176.772,8.547,148.751
C07937=1153.821,316.366,-74.844,-176.769,8.551,148.751
C07938=1153.817,316.613,-74.876,-176.767,8.554,148.751
C07939=1153.813,316.862,-74.907,-176.764,8.558,148.751
C07940=1153.809,317.110,-74.940,-176.762,8.561,148.752
C07941=1153.805,317.358,-74.972,-176.759,8.564,148.752
C07942=1153.801,317.605,-75.003,-176.756,8.568,148.752
C07943=1153.797,317.854,-75.036,-176.754,8.571,148.752
C07944=1153.793,318.102,-75.068,-176.751,8.575,148.752
C07945=1153.789,318.349,-75.099,-176.749,8.578,148.752
C07946=1153.784,318.597,-75.131,-176.746,8.582,148.753
C07947=1153.780,318.845,-75.163,-176.744,8.585,148.753
C07948=1153.776,319.093,-75.195,-176.741,8.588,148.753
C07949=1153.772,319.340,-75.228,-176.738,8.592,148.753
C07950=1153.768,319.588,-75.260,-176.736,8.596,148.753
C07951=1153.764,319.837,-75.292,-176.733,8.599,148.753
C07952=1153.759,320.084,-75.324,-176.731,8.602,148.754
C07953=1153.756,320.332,-75.356,-176.728,8.606,148.754
C07954=1153.751,320.581,-75.388,-176.725,8.609,148.754
C07955=1153.748,320.828,-75.421,-176.723,8.612,148.754
C07956=1153.743,321.076,-75.453,-176.720,8.617,148.754
C07957=1153.739,321.324,-75.484,-176.718,8.620,148.754
C07958=1153.735,321.572,-75.517,-176.716,8.623,148.755
C07959=1153.731,321.820,-75.549,-176.712,8.627,148.755
C07960=1153.727,322.068,-75.582,-176.710,8.630,148.755
C07961=1153.723,322.315,-75.613,-176.708,8.633,148.755
C07962=1153.718,322.563,-75.646,-176.705,8.637,148.755
C07963=1153.715,322.811,-75.678,-176.702,8.641,148.755
C07964=1153.710,323.059,-75.711,-176.700,8.644,148.756
C07965=1153.707,323.307,-75.743,-176.698,8.647,148.756
C07966=1153.702,323.556,-75.775,-176.694,8.651,148.756
C07967=1153.698,323.802,-75.807,-176.692,8.654,148.756
C07968=1153.694,324.051,-75.840,-176.690,8.658,148.756
C07969=1153.690,324.298,-75.872,-176.687,8.662,148.757
C07970=1153.686,324.546,-75.905,-176.685,8.665,148.757
C07971=1153.682,324.795,-75.937,-176.682,8.668,148.757
C07972=1153.678,325.042,-75.970,-176.679,8.672,148.757
C07973=1153.673,325.290,-76.002,-176.677,8.676,148.757
C07974=1153.670,325.537,-76.034,-176.674,8.679,148.757
C07975=1153.665,325.786,-76.067,-176.671,8.683,148.758
C07976=1153.662,326.033,-76.099,-176.669,8.686,148.758
C07977=1153.657,326.281,-76.132,-176.667,8.689,148.758
C07978=1153.653,326.529,-76.165,-176.664,8.693,148.758
C07979=1153.649,326.777,-76.197,-176.662,8.697,148.758
C07980=1153.645,327.025,-76.230,-176.659,8.700,148.759
C07981=1153.640,327.273,-76.262,-176.656,8.704,148.759
C07982=1153.637,327.520,-76.295,-176.654,8.707,148.759
C07983=1153.632,327.768,-76.327,-176.652,8.711,148.759
C07984=1153.628,328.016,-76.360,-176.649,8.715,148.759
C07985=1153.625,328.263,-76.393,-176.647,8.718,148.760
C07986=1153.620,328.512,-76.425,-176.644,8.721,148.760
C07987=1153.616,328.760,-76.458,-176.641,8.725,148.760
C07988=1153.612,329.007,-76.492,-176.639,8.728,148.760
C07989=1153.608,329.255,-76.523,-176.636,8.732,148.760
C07990=1153.604,329.503,-76.557,-176.633,8.736,148.760
C07991=1153.600,329.751,-76.590,-176.631,8.739,148.761
C07992=1153.596,329.999,-76.622,-176.628,8.743,148.761
C07993=1153.592,330.247,-76.655,-176.626,8.746,148.761
C07994=1153.588,330.494,-76.688,-176.624,8.750,148.761
C07995=1153.584,330.742,-76.721,-176.621,8.754,148.762
C07996=1153.580,330.990,-76.753,-176.618,8.757,148.762
C07997=1153.575,331.238,-76.787,-176.616,8.760,148.762
C07998=1153.572,331.486,-76.819,-176.613,8.764,148.762
C07999=1153.568,331.733,-76.852,-176.611,8.768,148.762
C08000=1153.563,331.982,-76.885,-176.608,8.772,148.763
C08001=1153.559,332.229,-76.918,-176.606,8.775,148.763
C08002=1153.555,332.477,-76.951,-176.603,8.778,148.763
C08003=1153.551,332.725,-76.984,-176.600,8.782,148.763
C08004=1153.547,332.973,-77.017,-176.598,8.786,148.763
C08005=1153.543,333.220,-77.051,-176.596,8.789,148.764
C08006=1153.539,333.468,-77.083,-176.593,8.793,148.764
C08007=1153.535,333.715,-77.116,-176.591,8.796,148.764
C08008=1153.531,333.963,-77.149,-176.588,8.800,148.764
C08009=1153.527,334.211,-77.183,-176.585,8.804,148.765
C08010=1153.523,334.459,-77.216,-176.583,8.807,148.765
C08011=1153.518,334.707,-77.248,-176.580,8.811,148.765
C08012=1153.514,334.955,-77.281,-176.578,8.814,148.765
C08013=1153.510,335.202,-77.314,-176.575,8.818,148.765
C08014=1153.506,335.449,-77.348,-176.573,8.822,148.766
C08015=1153.502,335.697,-77.381,-176.570,8.825,148.766
C08016=1153.498,335.945,-77.415,-176.567,8.829,148.766
C08017=1153.494,336.193,-77.448,-176.565,8.832,148.766
C08018=1153.490,336.440,-77.481,-176.563,8.836,148.767
C08019=1153.486,336.689,-77.514,-176.560,8.840,148.767
C08020=1153.482,336.937,-77.548,-176.558,8.843,148.767
C08021=1153.478,337.184,-77.581,-176.555,8.847,148.767
C08022=1153.474,337.432,-77.614,-176.552,8.850,148.767
C08023=1153.470,337.680,-77.647,-176.549,8.854,148.768
C08024=1153.466,337.927,-77.681,-176.548,8.858,148.768
C08025=1153.462,338.175,-77.714,-176.545,8.861,148.768
C08026=1153.458,338.422,-77.747,-176.542,8.865,148.769
C08027=1153.454,338.671,-77.781,-176.540,8.869,148.769
C08028=1153.450,338.918,-77.814,-176.537,8.873,148.769
C08029=1153.445,339.198,-77.852,-176.534,8.877,148.769
C08030=1153.441,339.479,-77.890,-176.531,8.881,148.769
C08031=1153.436,339.758,-77.927,-176.528,8.885,148.770
C08032=1153.431,340.039,-77.966,-176.525,8.889,148.770
C08033=1153.427,340.287,-77.999,-176.523,8.892,148.770
C08034=1153.423,340.534,-78.033,-176.521,8.897,148.771
C08035=1153.419,340.781,-78.066,-176.518,8.900,148.771
C08036=1153.415,341.029,-78.099,-176.516,8.903,148.771
C08037=1153.411,341.276,-78.133,-176.513,8.908,148.771
C08038=1153.407,341.525,-78.167,-176.511,8.911,148.771
C08039=1153.403,341.772,-78.201,-176.508,8.915,148.772
C08040=1153.399,342.020,-78.234,-176.506,8.918,148.772
C08041=1153.395,342.268,-78.267,-176.503,8.922,148.772
C08042=1153.391,342.516,-78.302,-176.500,8.926,148.772
C08043=1153.387,342.763,-78.335,-176.499,8.929,148.773
C08044=1153.383,343.011,-78.369,-176.496,8.933,148.773
C08045=1153.379,343.258,-78.403,-176.493,8.937,148.773
C08046=1153.374,343.506,-78.437,-176.490,8.941,148.774
C08047=1153.371,343.754,-78.471,-176.488,8.944,148.774
C08048=1153.367,344.001,-78.504,-176.485,8.948,148.774
C08049=1153.363,344.249,-78.538,-176.483,8.952,148.774
C08050=1153.358,344.496,-78.572,-176.480,8.956,148.775
C08051=1153.354,344.745,-78.606,-176.478,8.959,148.775
C08052=1153.351,344.992,-78.639,-176.475,8.963,148.775
C08053=1153.346,345.240,-78.673,-176.473,8.966,148.775
C08054=1153.343,345.488,-78.707,-176.470,8.970,148.776
C08055=1153.339,345.735,-78.741,-176.468,8.974,148.776
C08056=1153.334,345.983,-78.775,-176.466,8.977,148.776
C08057=1153.330,346.230,-78.809,-176.463,8.981,148.776
C08058=1153.327,346.478,-78.843,-176.461,8.985,148.777
C08059=1153.322,346.726,-78.877,-176.458,8.989,148.777
C08060=1153.318,346.973,-78.911,-176.456,8.992,148.777
C08061=1153.314,347.221,-78.946,-176.453,8.996,148.778
C08062=1153.310,347.469,-78.979,-176.451,9.000,148.778
C08063=1153.306,347.716,-79.013,-176.448,9.004,148.778
C08064=1153.302,347.964,-79.047,-176.445,9.007,148.778
C08065=1153.298,348.211,-79.081,-176.443,9.011,148.779
C08066=1153.293,348.459,-79.115,-176.441,9.015,148.779
C08067=1153.290,348.707,-79.149,-176.438,9.019,148.779
C08068=1153.286,348.954,-79.184,-176.435,9.022,148.779
C08069=1153.282,349.202,-79.218,-176.433,9.027,148.780
C08070=1153.278,349.450,-79.252,-176.431,9.030,148.780
C08071=1153.274,349.697,-79.286,-176.428,9.034,148.780
C08072=1153.270,349.946,-79.320,-176.425,9.037,148.780
C08073=1153.266,350.193,-79.354,-176.422,9.041,148.781
C08074=1153.262,350.441,-79.389,-176.421,9.045,148.781
C08075=1153.258,350.688,-79.423,-176.418,9.049,148.781
C08076=1153.254,350.935,-79.457,-176.415,9.052,148.782
C08077=1153.250,351.183,-79.492,-176.413,9.057,148.782
C08078=1153.246,351.430,-79.526,-176.411,9.060,148.782
C08079=1153.242,351.678,-79.560,-176.408,9.064,148.783
C08080=1153.238,351.926,-79.595,-176.405,9.067,148.783
C08081=1153.235,352.174,-79.629,-176.403,9.072,148.783
C08082=1153.230,352.421,-79.664,-176.401,9.075,148.783
C08083=1153.226,352.668,-79.698,-176.398,9.079,148.784
C08084=1153.222,352.916,-79.732,-176.395,9.082,148.784
C08085=1153.218,353.164,-79.767,-176.393,9.087,148.784
C08086=1153.215,353.411,-79.801,-176.391,9.090,148.785
C08087=1153.210,353.659,-79.835,-176.388,9.094,148.785
C08088=1153.206,353.907,-79.870,-176.385,9.099,148.785
C08089=1153.202,354.154,-79.904,-176.383,9.102,148.785
C08090=1153.198,354.402,-79.940,-176.380,9.106,148.786
C08091=1153.194,354.649,-79.974,-176.378,9.109,148.786
C08092=1153.191,354.897,-80.008,-176.375,9.114,148.786
C08093=1153.186,355.144,-80.043,-176.373,9.117,148.787
C08094=1153.182,355.392,-80.078,-176.370,9.121,148.787
C08095=1153.178,355.639,-80.112,-176.368,9.125,148.787
C08096=1153.175,355.887,-80.147,-176.365,9.129,148.788
C08097=1153.170,356.134,-80.182,-176.363,9.132,148.788
C08098=1153.167,356.382,-80.216,-176.360,9.136,148.788
C08099=1153.162,356.630,-80.250,-176.358,9.140,148.788
C08100=1153.159,356.877,-80.286,-176.356,9.144,148.789
C08101=1153.155,357.125,-80.321,-176.353,9.148,148.789
C08102=1153.151,357.372,-80.355,-176.350,9.151,148.789
C08103=1153.147,357.620,-80.390,-176.348,9.156,148.790
C08104=1153.143,357.867,-80.425,-176.346,9.159,148.790
C08105=1153.139,358.115,-80.459,-176.343,9.163,148.790
C08106=1153.135,358.362,-80.494,-176.341,9.167,148.791
C08107=1153.131,358.610,-80.529,-176.338,9.171,148.791
C08108=1153.127,358.858,-80.564,-176.335,9.175,148.791
C08109=1153.123,359.105,-80.599,-176.333,9.178,148.792
C08110=1153.119,359.353,-80.634,-176.330,9.183,148.792
C08111=1153.115,359.600,-80.669,-176.327,9.187,148.792
C08112=1153.111,359.848,-80.703,-176.325,9.190,148.793
C08113=1153.108,360.095,-80.739,-176.323,9.194,148.793
C08114=1153.103,360.343,-80.773,-176.320,9.198,148.793
C08115=1153.100,360.590,-80.809,-176.318,9.202,148.794
C08116=1153.096,360.838,-80.843,-176.315,9.206,148.794
C08117=1153.091,361.085,-80.879,-176.313,9.209,148.794
C08118=1153.087,361.333,-80.913,-176.310,9.214,148.795
C08119=1153.084,361.580,-80.948,-176.307,9.218,148.795
C08120=1153.080,361.828,-80.983,-176.305,9.221,148.795
C08121=1153.076,362.075,-81.018,-176.302,9.226,148.795
C08122=1153.073,362.323,-81.054,-176.299,9.230,148.796
C08123=1153.068,362.570,-81.088,-176.298,9.233,148.796
C08124=1153.064,362.818,-81.124,-176.295,9.237,148.796
C08125=1153.061,363.065,-81.160,-176.292,9.242,148.797
C08126=1153.056,363.313,-81.194,-176.290,9.245,148.797
C08127=1153.052,363.560,-81.230,-176.287,9.249,148.797
C08128=1153.049,363.808,-81.265,-176.285,9.254,148.798
C08129=1153.045,364.056,-81.300,-176.282,9.257,148.798
C08130=1153.040,364.302,-81.335,-176.280,9.261,148.799
C08131=1153.037,364.550,-81.371,-176.277,9.265,148.799
C08132=1153.033,364.797,-81.406,-176.275,9.269,148.799
C08133=1153.028,365.081,-81.446,-176.271,9.274,148.800
C08134=1153.024,365.364,-81.486,-176.269,9.278,148.800
C08135=1153.019,365.646,-81.527,-176.265,9.283,148.800
C08136=1153.015,365.930,-81.567,-176.263,9.288,148.801
C08137=1153.011,366.177,-81.603,-176.260,9.292,148.801
C08138=1153.007,366.425,-81.638,-176.258,9.295,148.802
C08139=1153.003,366.672,-81.674,-176.255,9.299,148.802
C08140=1152.999,366.919,-81.709,-176.253,9.304,148.802
C08141=1152.996,367.167,-81.745,-176.251,9.307,148.803
C08142=1152.992,367.414,-81.780,-176.248,9.311,148.803
C08143=1152.987,367.661,-81.816,-176.246,9.316,148.803
C08144=1152.983,367.909,-81.851,-176.243,9.319,148.804
C08145=1152.980,368.157,-81.886,-176.241,9.323,148.804
C08146=1152.976,368.404,-81.922,-176.238,9.328,148.805
C08147=1152.972,368.652,-81.958,-176.236,9.331,148.805
C08148=1152.969,368.899,-81.993,-176.234,9.336,148.805
C08149=1152.964,369.146,-82.029,-176.231,9.340,148.806
C08150=1152.960,369.394,-82.064,-176.229,9.344,148.806
C08151=1152.956,369.641,-82.100,-176.226,9.348,148.806
C08152=1152.953,369.888,-82.136,-176.224,9.352,148.807
C08153=1152.948,370.136,-82.172,-176.222,9.356,148.807
C08154=1152.945,370.384,-82.208,-176.219,9.360,148.808
C08155=1152.941,370.630,-82.243,-176.217,9.364,148.808
C08156=1152.937,370.878,-82.279,-176.215,9.368,148.809
C08157=1152.932,371.126,-82.315,-176.212,9.372,148.809
C08158=1152.929,371.373,-82.350,-176.210,9.376,148.809
C08159=1152.925,371.621,-82.386,-176.208,9.380,148.810
C08160=1152.922,371.868,-82.422,-176.205,9.384,148.810
C08161=1152.917,372.115,-82.458,-176.203,9.388,148.811
C08162=1152.914,372.363,-82.494,-176.201,9.392,148.811
C08163=1152.909,372.610,-82.529,-176.198,9.397,148.812
C08164=1152.905,372.858,-82.565,-176.197,9.401,148.812
C08165=1152.902,373.104,-82.601,-176.195,9.405,148.813
C08166=1152.898,373.352,-82.637,-176.193,9.409,148.813
C08167=1152.894,373.600,-82.673,-176.190,9.413,148.814
C08168=1152.890,373.847,-82.709,-176.188,9.417,148.814
C08169=1152.887,374.094,-82.745,-176.186,9.421,148.815
C08170=1152.882,374.342,-82.781,-176.184,9.425,148.815
C08171=1152.879,374.589,-82.817,-176.182,9.429,148.816
C08172=1152.875,374.836,-82.853,-176.180,9.433,148.816
C08173=1152.871,375.084,-82.889,-176.178,9.437,148.817
C08174=1152.867,375.331,-82.925,-176.176,9.442,148.817
C08175=1152.863,375.579,-82.961,-176.175,9.445,148.818
C08176=1152.859,375.826,-82.997,-176.172,9.450,148.818
C08177=1152.856,376.073,-83.033,-176.171,9.453,148.819
C08178=1152.852,376.321,-83.069,-176.169,9.457,148.820
C08179=1152.848,376.568,-83.106,-176.167,9.462,148.820
C08180=1152.844,376.816,-83.142,-176.165,9.466,148.821
C08181=1152.840,377.063,-83.178,-176.164,9.470,148.821
C08182=1152.836,377.310,-83.214,-176.162,9.473,148.822
C08183=1152.832,377.557,-83.250,-176.160,9.478,148.822
C08184=1152.828,377.804,-83.286,-176.158,9.482,148.823
C08185=1152.824,378.051,-83.322,-176.157,9.486,148.824
C08186=1152.821,378.300,-83.359,-176.155,9.490,148.824
C08187=1152.817,378.547,-83.395,-176.154,9.493,148.825
C08188=1152.813,378.795,-83.431,-176.152,9.497,148.825
C08189=1152.809,379.041,-83.468,-176.151,9.501,148.826
C08190=1152.805,379.289,-83.504,-176.149,9.505,148.827
C08191=1152.802,379.536,-83.540,-176.148,9.509,148.827
C08192=1152.798,379.783,-83.577,-176.147,9.513,148.828
C08193=1152.794,380.031,-83.612,-176.145,9.517,148.829
C08194=1152.790,380.278,-83.649,-176.144,9.521,148.829
C08195=1152.785,380.526,-83.685,-176.143,9.525,148.830
C08196=1152.782,380.773,-83.722,-176.141,9.529,148.831
C08197=1152.778,381.020,-83.759,-176.140,9.533,148.831
C08198=1152.774,381.267,-83.794,-176.139,9.536,148.832
C08199=1152.770,381.515,-83.831,-176.138,9.540,148.833
C08200=1152.766,381.762,-83.868,-176.137,9.544,148.833
C08201=1152.763,382.009,-83.904,-176.136,9.548,148.834
C08202=1152.758,382.256,-83.940,-176.135,9.552,148.835
C08203=1152.755,382.503,-83.977,-176.134,9.555,148.836
C08204=1152.751,382.750,-84.013,-176.133,9.559,148.836
C08205=1152.747,382.998,-84.050,-176.133,9.562,148.837
C08206=1152.744,383.246,-84.086,-176.132,9.567,148.838
C08207=1152.740,383.493,-84.123,-176.131,9.570,148.838
C08208=1152.736,383.740,-84.159,-176.130,9.573,148.839
C08209=1152.732,383.988,-84.195,-176.129,9.577,148.840
C08210=1152.728,384.235,-84.232,-176.129,9.581,148.841
C08211=1152.724,384.482,-84.269,-176.128,9.584,148.842
C08212=1152.720,384.729,-84.305,-176.128,9.587,148.842
C08213=1152.716,384.976,-84.342,-176.128,9.591,148.843
C08214=1152.713,385.224,-84.378,-176.127,9.594,148.844
C08215=1152.709,385.471,-84.415,-176.127,9.598,148.845
C08216=1152.705,385.719,-84.452,-176.126,9.601,148.846
C08217=1152.702,385.966,-84.488,-176.126,9.605,148.846
C08218=1152.698,386.213,-84.525,-176.126,9.607,148.847
C08219=1152.693,386.460,-84.562,-176.126,9.611,148.848
C08220=1152.689,386.708,-84.598,-176.126,9.614,148.849
C08221=1152.686,386.955,-84.634,-176.126,9.617,148.850
C08222=1152.682,387.202,-84.671,-176.126,9.620,148.850
C08223=1152.678,387.450,-84.708,-176.126,9.623,148.851
C08224=1152.675,387.697,-84.745,-176.126,9.627,148.852
C08225=1152.671,387.944,-84.781,-176.126,9.630,148.853
C08226=1152.667,388.191,-84.818,-176.126,9.632,148.854
C08227=1152.663,388.438,-84.855,-176.126,9.636,148.855
C08228=1152.659,388.685,-84.891,-176.126,9.638,148.855
C08229=1152.655,388.933,-84.928,-176.127,9.641,148.856
C08230=1152.651,389.181,-84.965,-176.127,9.644,148.857
C08231=1152.648,389.428,-85.001,-176.127,9.648,148.858
C08232=1152.644,389.675,-85.038,-176.128,9.650,148.859
C08233=1152.640,389.922,-85.075,-176.128,9.653,148.860
C08234=1152.636,390.169,-85.111,-176.128,9.656,148.860
C08235=1152.632,390.416,-85.148,-176.129,9.659,148.861
C08236=1152.628,390.663,-85.185,-176.129,9.662,148.862
C08237=1152.624,390.950,-85.227,-176.130,9.664,148.863
C08238=1152.620,391.236,-85.270,-176.131,9.668,148.864
C08239=1152.615,391.523,-85.313,-176.131,9.671,148.865
C08240=1152.611,391.808,-85.355,-176.132,9.673,148.866
C08241=1152.606,392.056,-85.391,-176.132,9.676,148.867
C08242=1152.603,392.304,-85.428,-176.133,9.679,148.868
C08243=1152.599,392.551,-85.465,-176.134,9.681,148.869
C08244=1152.595,392.798,-85.502,-176.134,9.684,148.869
C08245=1152.591,393.045,-85.539,-176.135,9.687,148.870
C08246=1152.588,393.292,-85.575,-176.136,9.689,148.871
C08247=1152.584,393.540,-85.612,-176.136,9.692,148.872
C08248=1152.580,393.787,-85.649,-176.137,9.694,148.873
C08249=1152.576,394.035,-85.686,-176.138,9.697,148.874
C08250=1152.573,394.281,-85.722,-176.139,9.698,148.874
C08251=1152.569,394.529,-85.759,-176.139,9.701,148.875
C08252=1152.565,394.776,-85.796,-176.140,9.703,148.876
C08253=1152.560,395.023,-85.833,-176.141,9.706,148.877
C08254=1152.558,395.271,-85.869,-176.142,9.708,148.878
C08255=1152.554,395.518,-85.906,-176.143,9.710,148.879
C08256=1152.549,395.765,-85.943,-176.143,9.713,148.879
C08257=1152.545,396.012,-85.980,-176.144,9.715,148.880
C08258=1152.541,396.259,-86.017,-176.145,9.717,148.881
C08259=1152.538,396.506,-86.053,-176.146,9.720,148.882
C08260=1152.534,396.754,-86.090,-176.147,9.722,148.883
C08261=1152.530,397.001,-86.127,-176.148,9.724,148.883
C08262=1152.526,397.249,-86.164,-176.149,9.726,148.884
C08263=1152.523,397.495,-86.200,-176.149,9.729,148.885
C08264=1152.519,397.743,-86.237,-176.151,9.731,148.886
C08265=1152.515,397.990,-86.274,-176.152,9.733,148.887
C08266=1152.511,398.238,-86.311,-176.152,9.734,148.887
C08267=1152.507,398.485,-86.348,-176.153,9.736,148.888
C08268=1152.504,398.732,-86.384,-176.155,9.739,148.889
C08269=1152.500,398.979,-86.421,-176.155,9.741,148.890
C08270=1152.496,399.226,-86.458,-176.156,9.743,148.891
C08271=1152.492,399.474,-86.495,-176.157,9.745,148.892
C08272=1152.488,399.721,-86.532,-176.158,9.747,148.892
C08273=1152.485,399.968,-86.568,-176.159,9.749,148.893
C08274=1152.481,400.215,-86.605,-176.160,9.751,148.894
C08275=1152.476,400.462,-86.642,-176.161,9.753,148.895
C08276=1152.472,400.710,-86.679,-176.162,9.755,148.896
C08277=1152.469,400.958,-86.716,-176.163,9.757,148.896
C08278=1152.466,401.204,-86.752,-176.164,9.759,148.897
C08279=1152.461,401.452,-86.789,-176.165,9.761,148.898
C08280=1152.457,401.699,-86.826,-176.166,9.763,148.899
C08281=1152.453,401.946,-86.863,-176.167,9.765,148.899
C08282=1152.450,402.193,-86.899,-176.167,9.767,148.900
C08283=1152.446,402.441,-86.936,-176.169,9.769,148.901
C08284=1152.442,402.688,-86.973,-176.170,9.771,148.902
C08285=1152.438,402.935,-87.010,-176.170,9.772,148.902
C08286=1152.434,403.182,-87.047,-176.171,9.775,148.903
C08287=1152.431,403.429,-87.083,-176.172,9.776,148.904
C08288=1152.427,403.677,-87.120,-176.173,9.778,148.905
C08289=1152.423,403.924,-87.157,-176.174,9.780,148.905
C08290=1152.419,404.172,-87.194,-176.175,9.782,148.906
C08291=1152.415,404.419,-87.231,-176.176,9.784,148.907
C08292=1152.412,404.666,-87.267,-176.177,9.786,148.908
C08293=1152.408,404.913,-87.304,-176.177,9.788,148.908
C08294=1152.404,405.161,-87.341,-176.179,9.790,148.909
C08295=1152.400,405.408,-87.378,-176.179,9.792,148.910
C08296=1152.396,405.655,-87.415,-176.180,9.794,148.911
C08297=1152.392,405.902,-87.451,-176.181,9.795,148.911
C08298=1152.388,406.149,-87.488,-176.182,9.797,148.912
C08299=1152.385,406.397,-87.525,-176.183,9.799,148.913
C08300=1152.381,406.644,-87.562,-176.184,9.801,148.913
C08301=1152.377,406.891,-87.599,-176.185,9.803,148.914
C08302=1152.373,407.138,-87.635,-176.185,9.805,148.915
C08303=1152.369,407.385,-87.672,-176.186,9.806,148.915
C08304=1152.365,407.633,-87.709,-176.187,9.809,148.916
C08305=1152.362,407.881,-87.746,-176.188,9.810,148.917
C08306=1152.358,408.128,-87.783,-176.188,9.812,148.918
C08307=1152.354,408.375,-87.820,-176.190,9.814,148.918
C08308=1152.350,408.622,-87.856,-176.190,9.816,148.919
C08309=1152.346,408.869,-87.893,-176.191,9.818,148.920
C08310=1152.343,409.117,-87.930,-176.192,9.819,148.920
C08311=1152.338,409.364,-87.967,-176.193,9.821,148.921
C08312=1152.335,409.611,-88.004,-176.193,9.823,148.922
C08313=1152.331,409.858,-88.040,-176.194,9.825,148.922
C08314=1152.327,410.105,-88.077,-176.195,9.827,148.923
C08315=1152.323,410.353,-88.114,-176.196,9.829,148.924
C08316=1152.320,410.600,-88.152,-176.197,9.830,148.925
C08317=1152.316,410.847,-88.188,-176.197,9.832,148.925
C08318=1152.312,411.094,-88.225,-176.198,9.834,148.926
C08319=1152.308,411.341,-88.262,-176.199,9.836,148.927
C08320=1152.304,411.588,-88.299,-176.199,9.837,148.927
C08321=1152.300,411.836,-88.336,-176.200,9.840,148.928
C08322=1152.296,412.083,-88.373,-176.201,9.841,148.929
C08323=1152.293,412.330,-88.409,-176.202,9.843,148.929
C08324=1152.289,412.577,-88.446,-176.202,9.845,148.930
C08325=1152.285,412.825,-88.483,-176.203,9.847,148.931
C08326=1152.281,413.072,-88.520,-176.204,9.848,148.931
C08327=1152.277,413.320,-88.557,-176.204,9.850,148.932
C08328=1152.274,413.567,-88.593,-176.205,9.852,148.932
C08329=1152.270,413.814,-88.630,-176.205,9.854,148.933
C08330=1152.266,414.061,-88.667,-176.206,9.856,148.934
C08331=1152.262,414.308,-88.704,-176.207,9.858,148.934
C08332=1152.258,414.556,-88.741,-176.208,9.860,148.935
C08333=1152.254,414.803,-88.778,-176.208,9.862,148.936
C08334=1152.251,415.050,-88.814,-176.209,9.863,148.937
C08335=1152.248,415.297,-88.852,-176.210,9.865,148.937
C08336=1152.247,415.545,-88.888,-176.210,9.867,148.938
C08337=1152.245,415.757,-88.920,-176.211,9.868,148.938
C08338=1152.245,415.971,-88.951,-176.211,9.870,148.939
C08339=1152.246,416.184,-88.982,-176.212,9.872,148.939
C08340=1152.246,416.397,-89.013,-176.212,9.873,148.940
C08341=1152.248,416.610,-89.045,-176.213,9.875,148.940
C08342=1152.250,416.822,-89.076,-176.213,9.876,148.941
C08343=1152.252,417.035,-89.107,-176.213,9.878,148.941
C08344=1152.255,417.247,-89.138,-176.214,9.879,148.942
C08345=1151.835,417.250,-89.186,-176.216,9.890,148.946
C08346=1151.832,417.035,-89.155,-176.216,9.889,148.945
C08347=1151.829,416.820,-89.124,-176.215,9.888,148.944
C08348=1151.827,416.607,-89.092,-176.215,9.886,148.944
C08349=1151.825,416.392,-89.061,-176.214,9.885,148.944
C08350=1151.825,416.177,-89.030,-176.214,9.883,148.943
C08351=1151.825,415.963,-88.998,-176.213,9.882,148.943
C08352=1151.825,415.747,-88.966,-176.213,9.880,148.942
C08353=1151.826,415.533,-88.934,-176.212,9.878,148.941
C08354=1151.828,415.286,-88.898,-176.212,9.877,148.941
C08355=1151.830,415.039,-88.861,-176.212,9.874,148.940
C08356=1151.834,414.792,-88.824,-176.211,9.872,148.939
C08357=1151.837,414.544,-88.787,-176.210,9.870,148.939
C08358=1151.841,414.297,-88.750,-176.209,9.869,148.938
C08359=1151.845,414.050,-88.714,-176.209,9.867,148.937
C08360=1151.849,413.802,-88.677,-176.208,9.865,148.937
C08361=1151.853,413.555,-88.640,-176.207,9.863,148.936
C08362=1151.857,413.307,-88.603,-176.207,9.862,148.935
C08363=1151.860,413.060,-88.566,-176.206,9.859,148.935
C08364=1151.864,412.813,-88.530,-176.206,9.857,148.934
C08365=1151.868,412.566,-88.493,-176.205,9.855,148.933
C08366=1151.872,412.319,-88.456,-176.204,9.854,148.933
C08367=1151.876,412.071,-88.419,-176.203,9.852,148.932
C08368=1151.879,411.824,-88.382,-176.203,9.850,148.931
C08369=1151.883,411.578,-88.345,-176.202,9.848,148.931
C08370=1151.887,411.330,-88.308,-176.201,9.846,148.930
C08371=1151.891,411.083,-88.271,-176.201,9.845,148.929
C08372=1151.895,410.836,-88.234,-176.200,9.843,148.929
C08373=1151.899,410.588,-88.197,-176.199,9.841,148.928
C08374=1151.902,410.341,-88.161,-176.198,9.839,148.927
C08375=1151.906,410.094,-88.124,-176.197,9.837,148.927
C08376=1151.910,409.847,-88.087,-176.197,9.836,148.926
C08377=1151.914,409.600,-88.050,-176.196,9.834,148.925
C08378=1151.918,409.352,-88.013,-176.195,9.832,148.925
C08379=1151.921,409.105,-87.977,-176.194,9.830,148.924
C08380=1151.925,408.858,-87.940,-176.194,9.828,148.923
C08381=1151.930,408.610,-87.903,-176.193,9.826,148.922
C08382=1151.934,408.363,-87.866,-176.192,9.824,148.922
C08383=1151.937,408.115,-87.829,-176.191,9.823,148.921
C08384=1151.940,407.869,-87.793,-176.190,9.821,148.920
C08385=1151.945,407.621,-87.756,-176.189,9.819,148.920
C08386=1151.949,407.374,-87.719,-176.189,9.817,148.919
C08387=1151.953,407.127,-87.682,-176.188,9.815,148.918
C08388=1151.957,406.880,-87.645,-176.187,9.813,148.917
C08389=1151.960,406.632,-87.608,-176.186,9.812,148.917
C08390=1151.964,406.385,-87.572,-176.185,9.810,148.916
C08391=1151.968,406.138,-87.535,-176.184,9.808,148.915
C08392=1151.972,405.891,-87.498,-176.183,9.806,148.915
C08393=1151.976,405.643,-87.461,-176.183,9.804,148.914
C08394=1151.979,405.396,-87.424,-176.182,9.802,148.913
C08395=1151.983,405.149,-87.388,-176.181,9.800,148.912
C08396=1151.987,404.902,-87.350,-176.180,9.798,148.912
C08397=1151.991,404.655,-87.313,-176.179,9.796,148.911
C08398=1151.995,404.408,-87.276,-176.178,9.794,148.910
C08399=1151.998,404.160,-87.239,-176.177,9.793,148.909
C08400=1152.002,403.913,-87.203,-176.176,9.790,148.909
C08401=1152.006,403.666,-87.166,-176.175,9.790,148.908
C08402=1152.010,403.419,-87.129,-176.174,9.787,148.907
C08403=1152.014,403.171,-87.092,-176.173,9.786,148.907
C08404=1152.018,402.924,-87.055,-176.172,9.784,148.906
C08405=1152.021,402.677,-87.019,-176.171,9.782,148.905
C08406=1152.025,402.429,-86.982,-176.170,9.780,148.904
C08407=1152.029,402.182,-86.945,-176.169,9.778,148.903
C08408=1152.033,401.935,-86.908,-176.168,9.776,148.903
C08409=1152.037,401.688,-86.871,-176.167,9.774,148.902
C08410=1152.040,401.440,-86.835,-176.166,9.772,148.901
C08411=1152.044,401.193,-86.798,-176.165,9.770,148.900
C08412=1152.048,400.946,-86.761,-176.164,9.768,148.900
C08413=1152.052,400.699,-86.724,-176.163,9.766,148.899
C08414=1152.056,400.451,-86.687,-176.163,9.764,148.898
C08415=1152.060,400.205,-86.651,-176.161,9.762,148.897
C08416=1152.063,399.957,-86.614,-176.160,9.760,148.896
C08417=1152.067,399.710,-86.577,-176.160,9.758,148.896
C08418=1152.071,399.462,-86.540,-176.159,9.756,148.895
C08419=1152.075,399.215,-86.503,-176.158,9.754,148.894
C08420=1152.079,398.968,-86.467,-176.157,9.751,148.893
C08421=1152.082,398.720,-86.430,-176.156,9.750,148.893
C08422=1152.086,398.473,-86.393,-176.155,9.748,148.892
C08423=1152.090,398.226,-86.356,-176.154,9.746,148.891
C08424=1152.095,397.979,-86.319,-176.153,9.744,148.890
C08425=1152.098,397.732,-86.283,-176.152,9.741,148.889
C08426=1152.102,397.485,-86.246,-176.152,9.739,148.888
C08427=1152.106,397.237,-86.209,-176.151,9.737,148.888
C08428=1152.110,396.990,-86.172,-176.149,9.735,148.887
C08429=1152.114,396.742,-86.135,-176.148,9.733,148.886
C08430=1152.117,396.496,-86.099,-176.148,9.730,148.885
C08431=1152.121,396.248,-86.062,-176.147,9.728,148.884
C08432=1152.125,396.001,-86.025,-176.146,9.726,148.884
C08433=1152.129,395.753,-85.988,-176.145,9.724,148.883
C08434=1152.132,395.506,-85.952,-176.144,9.721,148.882
C08435=1152.136,395.259,-85.915,-176.143,9.719,148.881
C08436=1152.140,395.012,-85.878,-176.142,9.717,148.880
C08437=1152.144,394.765,-85.841,-176.142,9.714,148.879
C08438=1152.148,394.517,-85.804,-176.141,9.712,148.879
C08439=1152.151,394.270,-85.768,-176.140,9.709,148.878
C08440=1152.155,394.023,-85.731,-176.139,9.707,148.877
C08441=1152.159,393.776,-85.694,-176.139,9.705,148.876
C08442=1152.164,393.528,-85.657,-176.138,9.702,148.875
C08443=1152.167,393.282,-85.621,-176.137,9.700,148.874
C08444=1152.170,393.034,-85.583,-176.136,9.698,148.874
C08445=1152.174,392.787,-85.547,-176.136,9.695,148.873
C08446=1152.179,392.539,-85.510,-176.135,9.692,148.872
C08447=1152.183,392.292,-85.473,-176.134,9.690,148.871
C08448=1152.186,392.045,-85.437,-176.134,9.687,148.870
C08449=1152.190,391.798,-85.400,-176.134,9.685,148.869
C08450=1152.194,391.511,-85.357,-176.133,9.681,148.868
C08451=1152.199,391.225,-85.314,-176.132,9.679,148.867
C08452=1152.203,390.938,-85.272,-176.131,9.675,148.866
C08453=1152.208,390.652,-85.230,-176.131,9.673,148.865
C08454=1152.212,390.404,-85.193,-176.130,9.670,148.864
C08455=1152.215,390.158,-85.156,-176.130,9.667,148.864
C08456=1152.219,389.910,-85.120,-176.129,9.664,148.863
C08457=1152.223,389.663,-85.083,-176.129,9.661,148.862
C08458=1152.227,389.416,-85.046,-176.129,9.659,148.861
C08459=1152.230,389.169,-85.010,-176.128,9.656,148.860
C08460=1152.234,388.921,-84.972,-176.128,9.652,148.859
C08461=1152.238,388.674,-84.936,-176.128,9.650,148.859
C08462=1152.242,388.427,-84.899,-176.128,9.647,148.858
C08463=1152.246,388.180,-84.862,-176.127,9.644,148.857
C08464=1152.250,387.933,-84.826,-176.128,9.640,148.856
C08465=1152.254,387.686,-84.789,-176.127,9.638,148.855
C08466=1152.257,387.438,-84.753,-176.127,9.635,148.855
C08467=1152.261,387.190,-84.716,-176.127,9.631,148.854
C08468=1152.265,386.943,-84.679,-176.127,9.628,148.853
C08469=1152.269,386.696,-84.642,-176.127,9.625,148.852
C08470=1152.272,386.449,-84.606,-176.127,9.622,148.851
C08471=1152.277,386.202,-84.569,-176.127,9.619,148.850
C08472=1152.281,385.955,-84.532,-176.128,9.616,148.850
C08473=1152.284,385.708,-84.496,-176.128,9.612,148.849
C08474=1152.288,385.459,-84.459,-176.128,9.609,148.848
C08475=1152.292,385.212,-84.423,-176.129,9.605,148.847
C08476=1152.295,384.965,-84.386,-176.129,9.602,148.846
C08477=1152.299,384.718,-84.350,-176.130,9.599,148.846
C08478=1152.303,384.471,-84.313,-176.130,9.595,148.845
C08479=1152.307,384.223,-84.277,-176.131,9.592,148.844
C08480=1152.311,383.976,-84.240,-176.131,9.588,148.843
C08481=1152.315,383.729,-84.203,-176.131,9.585,148.843
C08482=1152.319,383.482,-84.167,-176.132,9.581,148.842
C08483=1152.322,383.234,-84.130,-176.133,9.577,148.841
C08484=1152.327,382.986,-84.094,-176.133,9.574,148.840
C08485=1152.330,382.739,-84.057,-176.134,9.570,148.840
C08486=1152.334,382.492,-84.021,-176.135,9.567,148.839
C08487=1152.337,382.245,-83.984,-176.136,9.563,148.838
C08488=1152.342,381.997,-83.948,-176.137,9.559,148.837
C08489=1152.346,381.750,-83.911,-176.138,9.555,148.837
C08490=1152.349,381.503,-83.875,-176.139,9.551,148.836
C08491=1152.354,381.256,-83.839,-176.140,9.548,148.835
C08492=1152.358,381.008,-83.802,-176.141,9.544,148.835
C08493=1152.361,380.762,-83.766,-176.143,9.540,148.834
C08494=1152.365,380.514,-83.730,-176.144,9.536,148.833
C08495=1152.369,380.267,-83.693,-176.145,9.532,148.833
C08496=1152.373,380.020,-83.657,-176.147,9.528,148.832
C08497=1152.376,379.771,-83.621,-176.148,9.524,148.831
C08498=1152.380,379.524,-83.584,-176.149,9.521,148.831
C08499=1152.383,379.277,-83.548,-176.151,9.517,148.830
C08500=1152.388,379.030,-83.511,-176.152,9.512,148.829
C08501=1152.392,378.782,-83.475,-176.154,9.508,148.829
C08502=1152.396,378.535,-83.439,-176.155,9.504,148.828
C08503=1152.400,378.288,-83.402,-176.157,9.501,148.828
C08504=1152.403,378.040,-83.367,-176.159,9.497,148.827
C08505=1152.407,377.793,-83.330,-176.160,9.493,148.826
C08506=1152.411,377.546,-83.293,-176.162,9.489,148.826
C08507=1152.415,377.298,-83.257,-176.164,9.484,148.825
C08508=1152.419,377.051,-83.221,-176.165,9.480,148.824
C08509=1152.423,376.804,-83.185,-176.167,9.477,148.824
C08510=1152.427,376.556,-83.149,-176.168,9.473,148.823
C08511=1152.431,376.309,-83.113,-176.170,9.468,148.823
C08512=1152.434,376.061,-83.077,-176.172,9.465,148.822
C08513=1152.438,375.815,-83.041,-176.174,9.461,148.822
C08514=1152.442,375.567,-83.005,-176.176,9.456,148.821
C08515=1152.445,375.320,-82.968,-176.178,9.453,148.821
C08516=1152.450,375.072,-82.932,-176.180,9.448,148.820
C08517=1152.454,374.825,-82.897,-176.182,9.444,148.820
C08518=1152.457,374.578,-82.861,-176.184,9.440,148.819
C08519=1152.462,374.331,-82.825,-176.186,9.436,148.819
C08520=1152.466,374.083,-82.789,-176.188,9.432,148.818
C08521=1152.470,373.836,-82.752,-176.190,9.428,148.818
C08522=1152.473,373.588,-82.717,-176.193,9.424,148.817
C08523=1152.477,373.341,-82.681,-176.194,9.420,148.817
C08524=1152.481,373.094,-82.644,-176.197,9.416,148.816
C08525=1152.485,372.846,-82.609,-176.199,9.412,148.816
C08526=1152.488,372.599,-82.573,-176.201,9.407,148.815
C08527=1152.493,372.351,-82.537,-176.203,9.404,148.815
C08528=1152.496,372.104,-82.501,-176.205,9.399,148.814
C08529=1152.500,371.856,-82.465,-176.208,9.395,148.814
C08530=1152.505,371.609,-82.429,-176.210,9.391,148.813
C08531=1152.508,371.362,-82.394,-176.212,9.387,148.813
C08532=1152.512,371.114,-82.358,-176.214,9.383,148.812
C08533=1152.515,370.867,-82.322,-176.217,9.379,148.812
C08534=1152.520,370.620,-82.286,-176.219,9.375,148.812
C08535=1152.524,370.372,-82.250,-176.221,9.371,148.811
C08536=1152.527,370.125,-82.215,-176.224,9.367,148.811
C08537=1152.531,369.877,-82.179,-176.226,9.362,148.810
C08538=1152.536,369.630,-82.143,-176.228,9.359,148.810
C08539=1152.540,369.383,-82.108,-176.231,9.355,148.810
C08540=1152.543,369.135,-82.072,-176.233,9.350,148.809
C08541=1152.547,368.888,-82.037,-176.235,9.347,148.809
C08542=1152.551,368.640,-82.001,-176.238,9.343,148.808
C08543=1152.555,368.392,-81.965,-176.241,9.338,148.808
C08544=1152.559,368.145,-81.930,-176.243,9.335,148.808
C08545=1152.563,367.898,-81.894,-176.246,9.331,148.807
C08546=1152.566,367.650,-81.859,-176.248,9.326,148.807
C08547=1152.570,367.403,-81.823,-176.250,9.322,148.806
C08548=1152.574,367.155,-81.788,-176.253,9.318,148.806
C08549=1152.578,366.909,-81.753,-176.255,9.314,148.806
C08550=1152.582,366.661,-81.716,-176.258,9.310,148.805
C08551=1152.586,366.413,-81.681,-176.260,9.306,148.805
C08552=1152.590,366.166,-81.645,-176.263,9.302,148.805
C08553=1152.594,365.919,-81.610,-176.265,9.298,148.804
C08554=1152.599,365.635,-81.570,-176.268,9.294,148.804
C08555=1152.602,365.352,-81.530,-176.271,9.289,148.803
C08556=1152.608,365.069,-81.489,-176.274,9.284,148.803
C08557=1152.612,364.786,-81.449,-176.277,9.280,148.803
C08558=1152.616,364.538,-81.413,-176.279,9.276,148.802
C08559=1152.620,364.292,-81.378,-176.282,9.272,148.802
C08560=1152.624,364.044,-81.342,-176.284,9.268,148.802
C08561=1152.627,363.796,-81.308,-176.287,9.264,148.801
C08562=1152.631,363.549,-81.272,-176.290,9.260,148.801
C08563=1152.635,363.302,-81.237,-176.292,9.256,148.801
C08564=1152.639,363.054,-81.202,-176.295,9.252,148.800
C08565=1152.643,362.806,-81.166,-176.297,9.248,148.800
C08566=1152.647,362.559,-81.131,-176.300,9.244,148.800
C08567=1152.651,362.311,-81.096,-176.302,9.240,148.799
C08568=1152.655,362.064,-81.061,-176.305,9.236,148.799
C08569=1152.659,361.817,-81.026,-176.308,9.232,148.799
C08570=1152.662,361.569,-80.991,-176.310,9.228,148.798
C08571=1152.666,361.322,-80.956,-176.313,9.224,148.798
C08572=1152.671,361.074,-80.921,-176.315,9.220,148.798
C08573=1152.674,360.827,-80.886,-176.317,9.217,148.797
C08574=1152.678,360.579,-80.851,-176.320,9.212,148.797
C08575=1152.683,360.332,-80.816,-176.323,9.209,148.797
C08576=1152.687,360.084,-80.781,-176.325,9.205,148.796
C08577=1152.690,359.836,-80.746,-176.328,9.201,148.796
C08578=1152.694,359.589,-80.712,-176.330,9.197,148.796
C08579=1152.698,359.342,-80.676,-176.333,9.193,148.795
C08580=1152.702,359.094,-80.642,-176.336,9.189,148.795
C08581=1152.706,358.847,-80.606,-176.338,9.186,148.795
C08582=1152.710,358.598,-80.571,-176.340,9.181,148.794
C08583=1152.714,358.351,-80.537,-176.343,9.178,148.794
C08584=1152.717,358.104,-80.502,-176.345,9.174,148.794
C08585=1152.722,357.856,-80.467,-176.348,9.169,148.793
C08586=1152.726,357.609,-80.432,-176.350,9.166,148.793
C08587=1152.730,357.361,-80.397,-176.353,9.162,148.793
C08588=1152.733,357.114,-80.363,-176.355,9.159,148.793
C08589=1152.737,356.866,-80.328,-176.358,9.154,148.792
C08590=1152.742,356.619,-80.293,-176.360,9.151,148.792
C08591=1152.746,356.371,-80.258,-176.363,9.147,148.792
C08592=1152.749,356.124,-80.224,-176.366,9.143,148.791
C08593=1152.753,355.876,-80.189,-176.368,9.139,148.791
C08594=1152.758,355.629,-80.154,-176.371,9.135,148.791
C08595=1152.761,355.381,-80.120,-176.373,9.132,148.790
C08596=1152.765,355.133,-80.086,-176.375,9.127,148.790
C08597=1152.769,354.885,-80.051,-176.378,9.124,148.790
C08598=1152.773,354.638,-80.015,-176.381,9.120,148.790
C08599=1152.777,354.391,-79.981,-176.382,9.116,148.789
C08600=1152.781,354.143,-79.947,-176.385,9.112,148.789
C08601=1152.785,353.895,-79.913,-176.388,9.109,148.789
C08602=1152.789,353.648,-79.878,-176.390,9.105,148.788
C08603=1152.793,353.400,-79.843,-176.393,9.100,148.788
C08604=1152.797,353.153,-79.810,-176.395,9.097,148.788
C08605=1152.801,352.905,-79.775,-176.398,9.093,148.787
C08606=1152.806,352.657,-79.740,-176.400,9.089,148.787
C08607=1152.809,352.410,-79.705,-176.403,9.085,148.787
C08608=1152.813,352.163,-79.671,-176.405,9.082,148.787
C08609=1152.816,351.915,-79.637,-176.408,9.078,148.786
C08610=1152.821,351.667,-79.602,-176.410,9.074,148.786
C08611=1152.824,351.420,-79.568,-176.413,9.070,148.786
C08612=1152.829,351.172,-79.534,-176.415,9.067,148.785
C08613=1152.834,350.924,-79.500,-176.418,9.063,148.785
C08614=1152.837,350.676,-79.465,-176.420,9.059,148.785
C08615=1152.841,350.429,-79.431,-176.423,9.055,148.785
C08616=1152.845,350.181,-79.397,-176.425,9.052,148.784
C08617=1152.849,349.934,-79.362,-176.428,9.048,148.784
C08618=1152.853,349.687,-79.328,-176.430,9.044,148.784
C08619=1152.857,349.438,-79.294,-176.433,9.040,148.783
C08620=1152.861,349.191,-79.260,-176.435,9.037,148.783
C08621=1152.865,348.943,-79.225,-176.438,9.033,148.783
C08622=1152.869,348.696,-79.192,-176.440,9.029,148.783
C08623=1152.874,348.448,-79.157,-176.443,9.025,148.782
C08624=1152.877,348.200,-79.123,-176.445,9.022,148.782
C08625=1152.881,347.953,-79.089,-176.448,9.018,148.782
C08626=1152.885,347.705,-79.055,-176.450,9.014,148.781
C08627=1152.889,347.457,-79.021,-176.453,9.010,148.781
C08628=1152.893,347.210,-78.987,-176.455,9.007,148.781
C08629=1152.897,346.963,-78.953,-176.458,9.003,148.781
C08630=1152.901,346.714,-78.919,-176.460,8.999,148.780
C08631=1152.905,346.467,-78.885,-176.463,8.995,148.780
C08632=1152.909,346.220,-78.851,-176.465,8.992,148.780
C08633=1152.913,345.971,-78.817,-176.468,8.988,148.780
C08634=1152.917,345.724,-78.783,-176.471,8.984,148.779
C08635=1152.921,345.477,-78.749,-176.473,8.980,148.779
C08636=1152.925,345.228,-78.715,-176.475,8.977,148.779
C08637=1152.929,344.981,-78.681,-176.478,8.973,148.778
C08638=1152.933,344.733,-78.648,-176.481,8.969,148.778
C08639=1152.938,344.486,-78.614,-176.484,8.965,148.778
C08640=1152.941,344.238,-78.579,-176.485,8.962,148.778
C08641=1152.945,343.990,-78.546,-176.488,8.958,148.777
C08642=1152.950,343.743,-78.512,-176.491,8.954,148.777
C08643=1152.953,343.494,-78.478,-176.493,8.951,148.777
C08644=1152.957,343.247,-78.444,-176.496,8.947,148.777
C08645=1152.961,343.000,-78.411,-176.498,8.944,148.776
C08646=1152.966,342.752,-78.377,-176.501,8.939,148.776
C08647=1152.970,342.504,-78.343,-176.503,8.936,148.776
C08648=1152.973,342.257,-78.309,-176.506,8.932,148.776
C08649=1152.977,342.009,-78.276,-176.508,8.929,148.775
C08650=1152.982,341.761,-78.242,-176.511,8.925,148.775
C08651=1152.986,341.514,-78.208,-176.513,8.921,148.775
C08652=1152.990,341.265,-78.175,-176.516,8.918,148.775
C08653=1152.993,341.018,-78.141,-176.519,8.914,148.774
C08654=1152.998,340.771,-78.108,-176.520,8.910,148.774
C08655=1153.002,340.522,-78.074,-176.523,8.906,148.774
C08656=1153.006,340.275,-78.040,-176.526,8.903,148.774
C08657=1153.010,340.028,-78.007,-176.529,8.899,148.773
C08658=1153.014,339.747,-77.969,-176.532,8.895,148.773
C08659=1153.020,339.467,-77.931,-176.534,8.891,148.773
C08660=1153.024,339.187,-77.893,-176.537,8.887,148.773
C08661=1153.028,338.908,-77.856,-176.540,8.882,148.772
C08662=1153.032,338.660,-77.823,-176.542,8.879,148.772
C08663=1153.036,338.411,-77.789,-176.545,8.875,148.772
C08664=1153.041,338.163,-77.755,-176.547,8.872,148.771
C08665=1153.045,337.916,-77.722,-176.550,8.868,148.771
C08666=1153.049,337.669,-77.688,-176.553,8.864,148.771
C08667=1153.053,337.421,-77.655,-176.555,8.861,148.771
C08668=1153.057,337.173,-77.622,-176.558,8.857,148.771
C08669=1153.061,336.925,-77.589,-176.560,8.853,148.770
C08670=1153.065,336.677,-77.555,-176.563,8.849,148.770
C08671=1153.069,336.429,-77.522,-176.565,8.846,148.770
C08672=1153.073,336.181,-77.489,-176.568,8.843,148.770
C08673=1153.077,335.934,-77.456,-176.570,8.839,148.769
C08674=1153.081,335.687,-77.422,-176.573,8.835,148.769
C08675=1153.085,335.439,-77.389,-176.576,8.831,148.769
C08676=1153.089,335.191,-77.356,-176.578,8.828,148.769
C08677=1153.093,334.943,-77.322,-176.580,8.825,148.769
C08678=1153.098,334.696,-77.289,-176.583,8.821,148.768
C08679=1153.102,334.448,-77.256,-176.585,8.817,148.768
C08680=1153.106,334.200,-77.223,-176.588,8.813,148.768
C08681=1153.109,333.953,-77.190,-176.590,8.810,148.768
C08682=1153.113,333.704,-77.157,-176.593,8.807,148.767
C08683=1153.117,333.456,-77.124,-176.596,8.802,148.767
C08684=1153.121,333.208,-77.091,-176.598,8.799,148.767
C08685=1153.126,332.961,-77.058,-176.600,8.796,148.767
C08686=1153.130,332.713,-77.025,-176.603,8.792,148.766
C08687=1153.134,332.465,-76.992,-176.605,8.788,148.766
C08688=1153.138,332.217,-76.959,-176.608,8.784,148.766
C08689=1153.142,331.970,-76.926,-176.611,8.781,148.766
C08690=1153.145,331.722,-76.893,-176.613,8.778,148.766
C08691=1153.150,331.474,-76.861,-176.616,8.774,148.765
C08692=1153.154,331.226,-76.827,-176.618,8.770,148.765
C08693=1153.158,330.978,-76.794,-176.621,8.766,148.765
C08694=1153.162,330.731,-76.761,-176.623,8.763,148.765
C08695=1153.166,330.483,-76.728,-176.626,8.760,148.765
C08696=1153.170,330.235,-76.696,-176.629,8.756,148.764
C08697=1153.174,329.987,-76.663,-176.631,8.753,148.764
C08698=1153.178,329.739,-76.630,-176.634,8.749,148.764
C08699=1153.183,329.492,-76.598,-176.637,8.745,148.764
C08700=1153.187,329.244,-76.565,-176.639,8.742,148.764
C08701=1153.191,328.997,-76.532,-176.641,8.739,148.763
C08702=1153.195,328.748,-76.499,-176.644,8.735,148.763
C08703=1153.200,328.501,-76.466,-176.646,8.731,148.763
C08704=1153.203,328.253,-76.434,-176.649,8.727,148.763
C08705=1153.207,328.005,-76.401,-176.652,8.724,148.763
C08706=1153.212,327.757,-76.368,-176.654,8.721,148.762
C08707=1153.215,327.510,-76.336,-176.657,8.717,148.762
C08708=1153.219,327.261,-76.303,-176.659,8.713,148.762
C08709=1153.224,327.014,-76.270,-176.661,8.710,148.762
C08710=1153.228,326.765,-76.238,-176.664,8.706,148.762
C08711=1153.231,326.518,-76.205,-176.667,8.703,148.761
C08712=1153.236,326.270,-76.173,-176.669,8.700,148.761
C08713=1153.240,326.023,-76.140,-176.672,8.696,148.761
C08714=1153.244,325.774,-76.108,-176.675,8.692,148.761
C08715=1153.248,325.527,-76.075,-176.677,8.689,148.761
C08716=1153.252,325.279,-76.043,-176.680,8.685,148.760
C08717=1153.256,325.031,-76.010,-176.682,8.682,148.760
C08718=1153.261,324.783,-75.977,-176.684,8.679,148.760
C08719=1153.265,324.536,-75.945,-176.687,8.674,148.760
C08720=1153.269,324.288,-75.913,-176.690,8.671,148.760
C08721=1153.273,324.039,-75.881,-176.692,8.668,148.759
C08722=1153.277,323.792,-75.848,-176.695,8.664,148.759
C08723=1153.281,323.544,-75.816,-176.698,8.661,148.759
C08724=1153.285,323.295,-75.783,-176.700,8.658,148.759
C08725=1153.289,323.049,-75.751,-176.703,8.653,148.759
C08726=1153.294,322.800,-75.719,-176.705,8.650,148.759
C08727=1153.297,322.552,-75.687,-176.707,8.647,148.758
C08728=1153.301,322.305,-75.654,-176.710,8.643,148.758
C08729=1153.305,322.056,-75.622,-176.713,8.640,148.758
C08730=1153.310,321.808,-75.590,-176.715,8.637,148.758
C08731=1153.314,321.561,-75.557,-176.718,8.633,148.758
C08732=1153.318,321.313,-75.525,-176.721,8.629,148.758
C08733=1153.322,321.065,-75.493,-176.723,8.626,148.757
C08734=1153.326,320.817,-75.461,-176.725,8.623,148.757
C08735=1153.331,320.569,-75.429,-176.728,8.619,148.757
C08736=1153.335,320.322,-75.396,-176.731,8.616,148.757
C08737=1153.338,320.074,-75.364,-176.733,8.612,148.757
C08738=1153.342,319.826,-75.332,-176.736,8.608,148.757
C08739=1153.347,319.578,-75.300,-176.738,8.605,148.756
C08740=1153.351,319.330,-75.268,-176.741,8.602,148.756
C08741=1153.355,319.082,-75.236,-176.744,8.598,148.756
C08742=1153.359,318.833,-75.204,-176.746,8.595,148.756
C08743=1153.363,318.586,-75.173,-176.749,8.591,148.756
C08744=1153.367,318.338,-75.139,-176.751,8.588,148.756
C08745=1153.371,318.090,-75.108,-176.754,8.584,148.755
C08746=1153.375,317.842,-75.076,-176.757,8.581,148.755
C08747=1153.380,317.595,-75.044,-176.759,8.578,148.755
C08748=1153.384,317.347,-75.012,-176.762,8.574,148.755
C08749=1153.387,317.099,-74.980,-176.764,8.570,148.755
C08750=1153.392,316.851,-74.948,-176.767,8.567,148.755
C08751=1153.396,316.603,-74.916,-176.769,8.564,148.755
C08752=1153.400,316.355,-74.884,-176.772,8.560,148.754
C08753=1153.404,316.107,-74.853,-176.775,8.557,148.754
C08754=1153.409,315.859,-74.821,-176.777,8.554,148.754
C08755=1153.413,315.611,-74.789,-176.780,8.550,148.754
C08756=1153.417,315.363,-74.758,-176.783,8.546,148.754
C08757=1153.421,315.115,-74.725,-176.785,8.543,148.754
C08758=1153.425,314.867,-74.693,-176.787,8.540,148.753
C08759=1153.429,314.619,-74.662,-176.791,8.536,148.753
C08760=1153.433,314.371,-74.630,-176.793,8.533,148.753
C08761=1153.438,314.123,-74.599,-176.795,8.530,148.753
C08762=1153.443,313.846,-74.563,-176.798,8.526,148.753
C08763=1153.447,313.568,-74.527,-176.801,8.522,148.753
C08764=1153.451,313.291,-74.492,-176.804,8.518,148.753
C08765=1153.456,313.014,-74.457,-176.807,8.514,148.752
C08766=1153.460,312.766,-74.425,-176.809,8.511,148.752
C08767=1153.465,312.518,-74.394,-176.812,8.507,148.752
C08768=1153.468,312.270,-74.362,-176.815,8.504,148.752
C08769=1153.473,312.021,-74.330,-176.817,8.501,148.752
C08770=1153.477,311.773,-74.299,-176.820,8.498,148.752
C08771=1153.481,311.525,-74.267,-176.823,8.494,148.752
C08772=1153.485,311.278,-74.236,-176.825,8.490,148.751
C08773=1153.489,311.029,-74.205,-176.828,8.487,148.751
C08774=1153.494,310.782,-74.173,-176.830,8.484,148.751
C08775=1153.497,310.534,-74.141,-176.833,8.480,148.751
C08776=1153.502,310.286,-74.110,-176.836,8.477,148.751
C08777=1153.506,310.038,-74.079,-176.838,8.474,148.751
C08778=1153.510,309.790,-74.048,-176.840,8.471,148.751
C08779=1153.514,309.542,-74.016,-176.844,8.467,148.751
C08780=1153.519,309.294,-73.984,-176.846,8.464,148.750
C08781=1153.523,309.046,-73.953,-176.848,8.460,148.750
C08782=1153.527,308.798,-73.921,-176.850,8.457,148.750
C08783=1153.531,308.550,-73.890,-176.854,8.453,148.750
C08784=1153.536,308.302,-73.859,-176.856,8.450,148.750
C08785=1153.540,308.054,-73.828,-176.859,8.447,148.750
C08786=1153.544,307.806,-73.796,-176.861,8.444,148.750
C08787=1153.548,307.558,-73.765,-176.864,8.440,148.750
C08788=1153.553,307.310,-73.734,-176.867,8.437,148.750
C08789=1153.556,307.062,-73.702,-176.869,8.433,148.749
C08790=1153.561,306.814,-73.672,-176.871,8.430,148.749
C08791=1153.564,306.566,-73.640,-176.874,8.427,148.749
C08792=1153.568,306.318,-73.610,-176.877,8.423,148.749
C08793=1153.573,306.069,-73.578,-176.879,8.420,148.749
C08794=1153.577,305.822,-73.547,-176.882,8.417,148.749
C08795=1153.581,305.574,-73.516,-176.885,8.414,148.749
C08796=1153.585,305.325,-73.485,-176.887,8.410,148.748
C08797=1153.590,305.078,-73.454,-176.890,8.407,148.748
C08798=1153.594,304.829,-73.422,-176.893,8.403,148.748
C08799=1153.598,304.581,-73.392,-176.895,8.400,148.748
C08800=1153.602,304.333,-73.360,-176.898,8.397,148.748
C08801=1153.607,304.086,-73.329,-176.900,8.394,148.748
C08802=1153.611,303.838,-73.299,-176.903,8.390,148.748
C08803=1153.615,303.589,-73.268,-176.906,8.387,148.748
C08804=1153.619,303.342,-73.236,-176.908,8.384,148.748
C08805=1153.624,303.094,-73.206,-176.911,8.380,148.748
C08806=1153.628,302.845,-73.174,-176.913,8.377,148.747
C08807=1153.632,302.597,-73.144,-176.916,8.373,148.747
C08808=1153.635,302.349,-73.113,-176.919,8.370,148.747
C08809=1153.640,302.101,-73.082,-176.921,8.367,148.747
C08810=1153.644,301.854,-73.051,-176.924,8.364,148.747
C08811=1153.648,301.605,-73.020,-176.926,8.361,148.747
C08812=1153.653,301.357,-72.989,-176.929,8.357,148.747
C08813=1153.657,301.109,-72.959,-176.932,8.354,148.747
C08814=1153.661,300.861,-72.928,-176.934,8.351,148.747
C08815=1153.665,300.613,-72.897,-176.937,8.347,148.747
C08816=1153.670,300.365,-72.866,-176.940,8.344,148.747
C08817=1153.673,300.116,-72.836,-176.942,8.340,148.746
C08818=1153.678,299.868,-72.805,-176.945,8.337,148.746
C08819=1153.683,299.621,-72.774,-176.947,8.334,148.746
C08820=1153.686,299.373,-72.744,-176.950,8.331,148.746
C08821=1153.690,299.124,-72.713,-176.953,8.328,148.746
C08822=1153.695,298.876,-72.682,-176.955,8.325,148.746
C08823=1153.699,298.629,-72.652,-176.958,8.321,148.746
C08824=1153.703,298.380,-72.621,-176.961,8.318,148.746
C08825=1153.708,298.132,-72.590,-176.963,8.315,148.746
C08826=1153.711,297.884,-72.560,-176.966,8.311,148.746
C08827=1153.716,297.636,-72.529,-176.968,8.308,148.746
C08828=1153.720,297.388,-72.498,-176.971,8.305,148.745
C08829=1153.724,297.139,-72.468,-176.974,8.301,148.745
C08830=1153.729,296.892,-72.438,-176.976,8.298,148.745
C08831=1153.733,296.644,-72.408,-176.979,8.295,148.745
C08832=1153.737,296.395,-72.376,-176.981,8.292,148.745
C08833=1153.741,296.147,-72.346,-176.984,8.289,148.745
C08834=1153.745,295.900,-72.315,-176.986,8.286,148.745
C08835=1153.750,295.651,-72.285,-176.989,8.283,148.745
C08836=1153.753,295.403,-72.255,-176.992,8.279,148.745
C08837=1153.758,295.155,-72.224,-176.995,8.276,148.745
C08838=1153.762,294.907,-72.194,-176.997,8.272,148.745
C08839=1153.767,294.658,-72.164,-177.000,8.269,148.745
C08840=1153.771,294.411,-72.134,-177.003,8.266,148.745
C08841=1153.775,294.162,-72.103,-177.005,8.263,148.744
C08842=1153.779,293.914,-72.073,-177.008,8.259,148.744
C08843=1153.784,293.666,-72.042,-177.011,8.256,148.744
C08844=1153.787,293.418,-72.012,-177.013,8.253,148.744
C08845=1153.792,293.170,-71.982,-177.016,8.250,148.744
C08846=1153.796,292.922,-71.952,-177.019,8.247,148.744
C08847=1153.800,292.673,-71.921,-177.021,8.244,148.744
C08848=1153.804,292.425,-71.891,-177.024,8.241,148.744
C08849=1153.808,292.178,-71.861,-177.026,8.237,148.744
C08850=1153.813,291.929,-71.831,-177.029,8.234,148.744
C08851=1153.817,291.681,-71.801,-177.032,8.231,148.744
C08852=1153.822,291.433,-71.770,-177.034,8.227,148.744
C08853=1153.826,291.185,-71.741,-177.037,8.224,148.744
C08854=1153.829,290.937,-71.710,-177.039,8.221,148.744
C08855=1153.834,290.688,-71.680,-177.042,8.218,148.744
C08856=1153.838,290.440,-71.650,-177.045,8.215,148.743
C08857=1153.842,290.192,-71.621,-177.047,8.212,148.744
C08858=1153.847,289.944,-71.590,-177.051,8.208,148.744
C08859=1153.851,289.696,-71.560,-177.053,8.205,148.743
C08860=1153.856,289.448,-71.530,-177.056,8.202,148.743
C08861=1153.860,289.200,-71.500,-177.058,8.199,148.743
C08862=1153.864,288.952,-71.471,-177.061,8.196,148.743
C08863=1153.868,288.704,-71.441,-177.064,8.193,148.743
C08864=1153.872,288.455,-71.410,-177.066,8.190,148.743
C08865=1153.876,288.207,-71.380,-177.069,8.187,148.743
C08866=1153.881,287.932,-71.347,-177.072,8.183,148.743
C08867=1153.886,287.657,-71.314,-177.074,8.180,148.743
C08868=1153.890,287.381,-71.281,-177.078,8.176,148.743
C08869=1153.895,287.107,-71.248,-177.081,8.172,148.743
C08870=1153.900,286.858,-71.218,-177.083,8.169,148.743
C08871=1153.904,286.610,-71.189,-177.086,8.166,148.743
C08872=1153.908,286.362,-71.158,-177.088,8.163,148.743
C08873=1153.912,286.114,-71.129,-177.091,8.160,148.743
C08874=1153.917,285.865,-71.099,-177.094,8.157,148.743
C08875=1153.921,285.617,-71.069,-177.096,8.153,148.743
C08876=1153.925,285.369,-71.039,-177.099,8.150,148.743
C08877=1153.929,285.121,-71.010,-177.102,8.148,148.743
C08878=1153.934,284.873,-70.980,-177.104,8.144,148.743
C08879=1153.938,284.625,-70.951,-177.107,8.141,148.743
C08880=1153.943,284.376,-70.921,-177.110,8.137,148.742
C08881=1153.947,284.128,-70.891,-177.113,8.134,148.742
C08882=1153.951,283.880,-70.861,-177.115,8.131,148.742
C08883=1153.955,283.632,-70.832,-177.118,8.128,148.742
C08884=1153.959,283.384,-70.802,-177.120,8.125,148.742
C08885=1153.963,283.135,-70.773,-177.123,8.122,148.742
C08886=1153.967,282.887,-70.743,-177.125,8.119,148.742
C08887=1153.972,282.638,-70.713,-177.128,8.116,148.742
C08888=1153.977,282.390,-70.684,-177.131,8.113,148.742
C08889=1153.981,282.142,-70.655,-177.133,8.110,148.742
C08890=1153.985,281.894,-70.625,-177.136,8.107,148.742
C08891=1153.989,281.645,-70.596,-177.139,8.104,148.742
C08892=1153.993,281.397,-70.566,-177.142,8.101,148.742
C08893=1153.998,281.149,-70.537,-177.145,8.097,148.742
C08894=1154.002,280.901,-70.508,-177.147,8.094,148.742
C08895=1154.006,280.653,-70.478,-177.150,8.091,148.742
C08896=1154.011,280.405,-70.449,-177.152,8.088,148.742
C08897=1154.015,280.156,-70.419,-177.155,8.085,148.742
C08898=1154.019,279.908,-70.390,-177.158,8.082,148.742
C08899=1154.023,279.660,-70.360,-177.160,8.078,148.742
C08900=1154.027,279.412,-70.331,-177.163,8.075,148.742
C08901=1154.032,279.163,-70.302,-177.166,8.073,148.742
C08902=1154.037,278.915,-70.273,-177.169,8.070,148.742
C08903=1154.041,278.667,-70.244,-177.171,8.066,148.742
C08904=1154.045,278.419,-70.214,-177.174,8.063,148.742
C08905=1154.049,278.170,-70.185,-177.176,8.060,148.742
C08906=1154.053,277.922,-70.155,-177.179,8.057,148.742
C08907=1154.058,277.673,-70.127,-177.181,8.054,148.742
C08908=1154.062,277.425,-70.097,-177.184,8.051,148.742
C08909=1154.066,277.178,-70.069,-177.187,8.048,148.742
C08910=1154.070,276.929,-70.039,-177.190,8.045,148.742
C08911=1154.075,276.681,-70.010,-177.192,8.042,148.742
C08912=1154.079,276.432,-69.981,-177.195,8.038,148.742
C08913=1154.083,276.184,-69.951,-177.198,8.035,148.742
C08914=1154.088,275.936,-69.922,-177.201,8.032,148.742
C08915=1154.092,275.688,-69.894,-177.203,8.029,148.742
C08916=1154.096,275.440,-69.865,-177.206,8.026,148.742
C08917=1154.100,275.191,-69.835,-177.209,8.023,148.742
C08918=1154.104,274.942,-69.807,-177.212,8.020,148.742
C08919=1154.109,274.695,-69.778,-177.214,8.017,148.742
C08920=1154.113,274.447,-69.748,-177.217,8.014,148.742
C08921=1154.118,274.198,-69.719,-177.219,8.011,148.742
C08922=1154.121,273.950,-69.690,-177.222,8.008,148.742
C08923=1154.126,273.702,-69.662,-177.225,8.005,148.742
C08924=1154.131,273.453,-69.633,-177.227,8.002,148.742
C08925=1154.135,273.204,-69.604,-177.230,7.999,148.742
C08926=1154.139,272.956,-69.575,-177.233,7.996,148.742
C08927=1154.144,272.708,-69.547,-177.236,7.993,148.742
C08928=1154.148,272.460,-69.517,-177.238,7.990,148.742
C08929=1154.152,272.211,-69.488,-177.241,7.987,148.742
C08930=1154.156,271.964,-69.460,-177.243,7.984,148.742
C08931=1154.161,271.715,-69.431,-177.246,7.981,148.742
C08932=1154.165,271.467,-69.402,-177.249,7.978,148.742
C08933=1154.169,271.218,-69.374,-177.252,7.975,148.742
C08934=1154.174,270.971,-69.345,-177.254,7.972,148.742
C08935=1154.178,270.722,-69.316,-177.257,7.969,148.742
C08936=1154.182,270.474,-69.287,-177.260,7.966,148.742
C08937=1154.187,270.226,-69.259,-177.262,7.963,148.742
C08938=1154.191,269.977,-69.230,-177.265,7.960,148.742
C08939=1154.195,269.729,-69.201,-177.268,7.957,148.742
C08940=1154.200,269.481,-69.173,-177.270,7.954,148.742
C08941=1154.204,269.232,-69.144,-177.273,7.951,148.742
C08942=1154.208,268.984,-69.115,-177.276,7.948,148.742
C08943=1154.213,268.736,-69.087,-177.279,7.945,148.742
C08944=1154.216,268.487,-69.059,-177.281,7.942,148.742
C08945=1154.221,268.239,-69.030,-177.284,7.939,148.742
C08946=1154.226,267.990,-69.001,-177.286,7.936,148.742
C08947=1154.229,267.742,-68.973,-177.289,7.933,148.742
C08948=1154.235,267.494,-68.944,-177.292,7.930,148.742
C08949=1154.238,267.245,-68.916,-177.295,7.927,148.742
C08950=1154.243,266.998,-68.887,-177.297,7.924,148.742
C08951=1154.247,266.749,-68.859,-177.300,7.921,148.742
C08952=1154.251,266.500,-68.830,-177.303,7.918,148.742
C08953=1154.256,266.252,-68.802,-177.305,7.915,148.742
C08954=1154.260,266.003,-68.774,-177.308,7.912,148.742
C08955=1154.265,265.755,-68.745,-177.311,7.909,148.742
C08956=1154.269,265.507,-68.716,-177.314,7.906,148.742
C08957=1154.274,265.259,-68.688,-177.316,7.903,148.743
C08958=1154.277,265.010,-68.660,-177.319,7.900,148.743
C08959=1154.281,264.762,-68.632,-177.322,7.897,148.743
C08960=1154.286,264.514,-68.603,-177.325,7.894,148.743
C08961=1154.290,264.265,-68.575,-177.328,7.891,148.743
C08962=1154.295,264.017,-68.547,-177.330,7.888,148.743
C08963=1154.299,263.768,-68.519,-177.332,7.886,148.743
C08964=1154.304,263.520,-68.490,-177.335,7.883,148.743
C08965=1154.308,263.272,-68.462,-177.338,7.880,148.743
C08966=1154.313,263.023,-68.434,-177.340,7.877,148.743
C08967=1154.317,262.775,-68.406,-177.343,7.874,148.743
C08968=1154.321,262.527,-68.378,-177.346,7.871,148.743
C08969=1154.325,262.278,-68.349,-177.349,7.868,148.743
C08970=1154.330,262.005,-68.318,-177.352,7.865,148.743
C08971=1154.335,261.731,-68.288,-177.355,7.862,148.743
C08972=1154.339,261.458,-68.257,-177.358,7.859,148.743
C08973=1154.345,261.185,-68.225,-177.361,7.855,148.743
C08974=1154.349,260.937,-68.197,-177.364,7.852,148.743
C08975=1154.353,260.688,-68.170,-177.366,7.850,148.743
C08976=1154.358,260.440,-68.141,-177.369,7.847,148.743
C08977=1154.362,260.191,-68.113,-177.371,7.844,148.743
C08978=1154.366,259.943,-68.086,-177.374,7.841,148.744
C08979=1154.370,259.695,-68.057,-177.377,7.838,148.744
C08980=1154.375,259.447,-68.029,-177.380,7.835,148.744
C08981=1154.380,259.198,-68.002,-177.382,7.832,148.744
C08982=1154.383,258.949,-67.974,-177.385,7.829,148.744
C08983=1154.388,258.701,-67.945,-177.388,7.826,148.744
C08984=1154.392,258.453,-67.917,-177.390,7.823,148.744
C08985=1154.397,258.204,-67.890,-177.393,7.820,148.744
C08986=1154.401,257.956,-67.862,-177.396,7.817,148.744
C08987=1154.405,257.708,-67.834,-177.399,7.814,148.744
C08988=1154.410,257.459,-67.807,-177.401,7.811,148.744
C08989=1154.414,257.210,-67.779,-177.404,7.809,148.744
C08990=1154.418,256.963,-67.751,-177.406,7.806,148.744
C08991=1154.423,256.714,-67.724,-177.409,7.803,148.744
C08992=1154.427,256.465,-67.696,-177.412,7.800,148.744
C08993=1154.432,256.217,-67.667,-177.415,7.797,148.744
C08994=1154.436,255.968,-67.640,-177.418,7.794,148.744
C08995=1154.440,255.720,-67.612,-177.420,7.792,148.744
C08996=1154.445,255.472,-67.585,-177.423,7.789,148.744
C08997=1154.449,255.223,-67.557,-177.426,7.786,148.745
C08998=1154.453,254.975,-67.529,-177.429,7.783,148.745
C08999=1154.458,254.727,-67.502,-177.431,7.780,148.745
C09000=1154.462,254.478,-67.473,-177.434,7.778,148.745
C09001=1154.467,254.229,-67.446,-177.436,7.775,148.745
C09002=1154.471,253.981,-67.418,-177.439,7.772,148.745
C09003=1154.475,253.732,-67.391,-177.442,7.769,148.745
C09004=1154.480,253.484,-67.363,-177.445,7.766,148.745
C09005=1154.484,253.236,-67.336,-177.447,7.763,148.745
C09006=1154.488,252.987,-67.308,-177.450,7.760,148.745
C09007=1154.493,252.739,-67.281,-177.453,7.757,148.745
C09008=1154.497,252.490,-67.254,-177.456,7.754,148.745
C09009=1154.502,252.242,-67.226,-177.459,7.751,148.745
C09010=1154.506,251.993,-67.199,-177.461,7.749,148.745
C09011=1154.510,251.745,-67.171,-177.464,7.746,148.746
C09012=1154.515,251.497,-67.144,-177.466,7.743,148.746
C09013=1154.519,251.248,-67.116,-177.469,7.740,148.746
C09014=1154.523,251.000,-67.089,-177.472,7.737,148.746
C09015=1154.528,250.751,-67.062,-177.475,7.735,148.746
C09016=1154.533,250.503,-67.034,-177.478,7.732,148.746
C09017=1154.536,250.254,-67.006,-177.481,7.729,148.746
C09018=1154.541,250.006,-66.979,-177.483,7.727,148.746
C09019=1154.546,249.757,-66.952,-177.486,7.724,148.746
C09020=1154.550,249.509,-66.924,-177.488,7.721,148.746
C09021=1154.555,249.261,-66.897,-177.491,7.718,148.746
C09022=1154.559,249.012,-66.870,-177.494,7.715,148.747
C09023=1154.563,248.763,-66.843,-177.497,7.712,148.747
C09024=1154.567,248.515,-66.816,-177.499,7.709,148.747
C09025=1154.572,248.267,-66.789,-177.502,7.706,148.747
C09026=1154.576,248.019,-66.762,-177.504,7.704,148.747
C09027=1154.580,247.769,-66.734,-177.507,7.701,148.747
C09028=1154.585,247.521,-66.707,-177.510,7.698,148.747
C09029=1154.590,247.272,-66.680,-177.513,7.695,148.747
C09030=1154.594,247.024,-66.653,-177.516,7.693,148.747
C09031=1154.599,246.776,-66.625,-177.519,7.690,148.747
C09032=1154.603,246.528,-66.599,-177.521,7.688,148.748
C09033=1154.607,246.279,-66.571,-177.524,7.685,148.748
C09034=1154.611,246.030,-66.544,-177.527,7.682,148.748
C09035=1154.616,245.782,-66.517,-177.529,7.679,148.748
C09036=1154.621,245.533,-66.490,-177.532,7.676,148.748
C09037=1154.624,245.285,-66.464,-177.535,7.673,148.748
C09038=1154.629,245.037,-66.437,-177.538,7.670,148.748
C09039=1154.634,244.788,-66.410,-177.540,7.668,148.748
C09040=1154.638,244.539,-66.382,-177.543,7.665,148.748
C09041=1154.642,244.291,-66.356,-177.546,7.662,148.748
C09042=1154.646,244.042,-66.329,-177.549,7.659,148.748
C09043=1154.651,243.794,-66.301,-177.551,7.656,148.749
C09044=1154.656,243.545,-66.274,-177.554,7.653,148.749
C09045=1154.660,243.297,-66.248,-177.556,7.651,148.749
C09046=1154.664,243.048,-66.221,-177.559,7.648,148.749
C09047=1154.669,242.800,-66.194,-177.562,7.646,148.749
C09048=1154.673,242.552,-66.167,-177.565,7.643,148.749
C09049=1154.678,242.303,-66.140,-177.568,7.640,148.749
C09050=1154.682,242.053,-66.114,-177.570,7.638,148.749
C09051=1154.687,241.805,-66.087,-177.573,7.635,148.749
C09052=1154.690,241.557,-66.060,-177.576,7.632,148.749
C09053=1154.695,241.308,-66.033,-177.579,7.629,148.750
C09054=1154.699,241.060,-66.007,-177.581,7.626,148.750
C09055=1154.704,240.812,-65.979,-177.584,7.623,148.750
C09056=1154.709,240.563,-65.953,-177.587,7.621,148.750
C09057=1154.713,240.314,-65.927,-177.590,7.618,148.750
C09058=1154.717,240.066,-65.900,-177.592,7.616,148.750
C09059=1154.722,239.817,-65.873,-177.595,7.613,148.750
C09060=1154.726,239.569,-65.847,-177.598,7.610,148.750
C09061=1154.731,239.320,-65.820,-177.600,7.608,148.750
C09062=1154.735,239.072,-65.793,-177.603,7.605,148.751
C09063=1154.739,238.823,-65.766,-177.606,7.602,148.751
C09064=1154.744,238.575,-65.740,-177.609,7.599,148.751
C09065=1154.748,238.326,-65.713,-177.612,7.596,148.751
C09066=1154.753,238.078,-65.686,-177.614,7.594,148.751
C09067=1154.757,237.829,-65.661,-177.617,7.591,148.751
C09068=1154.762,237.580,-65.634,-177.620,7.588,148.751
C09069=1154.766,237.331,-65.608,-177.623,7.586,148.752
C09070=1154.771,237.083,-65.581,-177.625,7.583,148.752
C09071=1154.775,236.835,-65.554,-177.628,7.580,148.752
C09072=1154.780,236.586,-65.528,-177.630,7.578,148.752
C09073=1154.783,236.337,-65.501,-177.634,7.575,148.752
C09074=1154.789,236.065,-65.473,-177.636,7.572,148.752
C09075=1154.793,235.794,-65.444,-177.639,7.569,148.752
C09076=1154.798,235.522,-65.415,-177.642,7.567,148.753
C09077=1154.803,235.250,-65.387,-177.645,7.564,148.753
C09078=1154.808,235.002,-65.360,-177.648,7.561,148.753
C09079=1154.812,234.753,-65.334,-177.651,7.558,148.753
C09080=1154.817,234.505,-65.307,-177.654,7.555,148.753
C09081=1154.821,234.256,-65.281,-177.656,7.553,148.753
C09082=1154.825,234.008,-65.255,-177.659,7.550,148.753
C09083=1154.830,233.759,-65.229,-177.662,7.547,148.753
C09084=1154.834,233.511,-65.202,-177.665,7.544,148.753
C09085=1154.838,233.262,-65.176,-177.667,7.542,148.754
C09086=1154.843,233.013,-65.150,-177.670,7.539,148.754
C09087=1154.847,232.765,-65.124,-177.673,7.537,148.754
C09088=1154.852,232.516,-65.097,-177.676,7.534,148.754
C09089=1154.857,232.267,-65.071,-177.678,7.532,148.754
C09090=1154.861,232.020,-65.045,-177.681,7.529,148.754
C09091=1154.866,231.770,-65.019,-177.684,7.526,148.754
C09092=1154.870,231.522,-64.993,-177.687,7.523,148.755
C09093=1154.874,231.273,-64.967,-177.689,7.521,148.755
C09094=1154.878,231.025,-64.941,-177.692,7.518,148.755
C09095=1154.883,230.776,-64.915,-177.695,7.515,148.755
C09096=1154.888,230.528,-64.889,-177.698,7.512,148.755
C09097=1154.892,230.279,-64.863,-177.700,7.510,148.755
C09098=1154.897,230.030,-64.837,-177.703,7.508,148.756
C09099=1154.901,229.781,-64.811,-177.706,7.505,148.756
C09100=1154.905,229.533,-64.784,-177.709,7.502,148.756
C09101=1154.910,229.285,-64.759,-177.711,7.500,148.756
C09102=1154.915,229.036,-64.733,-177.714,7.497,148.756
C09103=1154.919,228.787,-64.707,-177.717,7.494,148.756
C09104=1154.923,228.538,-64.681,-177.719,7.492,148.756
C09105=1154.928,228.290,-64.655,-177.722,7.490,148.757
C09106=1154.932,228.042,-64.629,-177.725,7.487,148.757
C09107=1154.937,227.793,-64.603,-177.728,7.484,148.757
C09108=1154.941,227.544,-64.577,-177.730,7.482,148.757
C09109=1154.946,227.295,-64.551,-177.733,7.479,148.757
C09110=1154.950,227.047,-64.526,-177.736,7.476,148.757
C09111=1154.955,226.798,-64.500,-177.738,7.474,148.757
C09112=1154.959,226.550,-64.474,-177.742,7.471,148.758
C09113=1154.963,226.301,-64.449,-177.744,7.468,148.758
C09114=1154.969,226.052,-64.423,-177.747,7.466,148.758
C09115=1154.973,225.804,-64.397,-177.749,7.463,148.758
C09116=1154.977,225.555,-64.371,-177.753,7.461,148.758
C09117=1154.982,225.307,-64.346,-177.755,7.458,148.758
C09118=1154.986,225.058,-64.320,-177.758,7.456,148.759
C09119=1154.990,224.809,-64.294,-177.761,7.453,148.759
C09120=1154.995,224.560,-64.269,-177.764,7.450,148.759
C09121=1154.999,224.312,-64.243,-177.766,7.448,148.759
C09122=1155.004,224.063,-64.217,-177.769,7.446,148.759
C09123=1155.008,223.815,-64.192,-177.772,7.443,148.759
C09124=1155.013,223.566,-64.166,-177.774,7.440,148.760
C09125=1155.017,223.318,-64.141,-177.777,7.438,148.760
C09126=1155.021,223.069,-64.115,-177.780,7.435,148.760
C09127=1155.027,222.820,-64.090,-177.783,7.432,148.760
C09128=1155.031,222.571,-64.064,-177.785,7.430,148.760
C09129=1155.035,222.322,-64.038,-177.788,7.427,148.760
C09130=1155.040,222.074,-64.013,-177.791,7.424,148.761
C09131=1155.045,221.825,-63.987,-177.793,7.422,148.761
C09132=1155.048,221.577,-63.962,-177.797,7.420,148.761
C09133=1155.053,221.328,-63.937,-177.799,7.417,148.761
C09134=1155.057,221.079,-63.911,-177.801,7.415,148.761
C09135=1155.062,220.831,-63.886,-177.805,7.412,148.761
C09136=1155.066,220.582,-63.860,-177.807,7.410,148.762
C09137=1155.071,220.333,-63.835,-177.810,7.407,148.762
C09138=1155.076,220.085,-63.810,-177.813,7.404,148.762
C09139=1155.080,219.836,-63.784,-177.815,7.402,148.762
C09140=1155.085,219.588,-63.759,-177.818,7.400,148.762
C09141=1155.089,219.339,-63.734,-177.821,7.397,148.762
C09142=1155.094,219.090,-63.708,-177.823,7.395,148.763
C09143=1155.098,218.842,-63.682,-177.827,7.392,148.763
C09144=1155.102,218.592,-63.658,-177.829,7.389,148.763
C09145=1155.107,218.344,-63.633,-177.832,7.387,148.763
C09146=1155.111,218.096,-63.607,-177.835,7.385,148.763
C09147=1155.116,217.847,-63.582,-177.838,7.382,148.764
C09148=1155.121,217.598,-63.556,-177.840,7.379,148.764
C09149=1155.125,217.349,-63.531,-177.843,7.377,148.764
